REGION Network 9: Make Up Spin
   // Output if Throttle not disabled after a shift, flush not disabled, Drill Throttle Input Zero
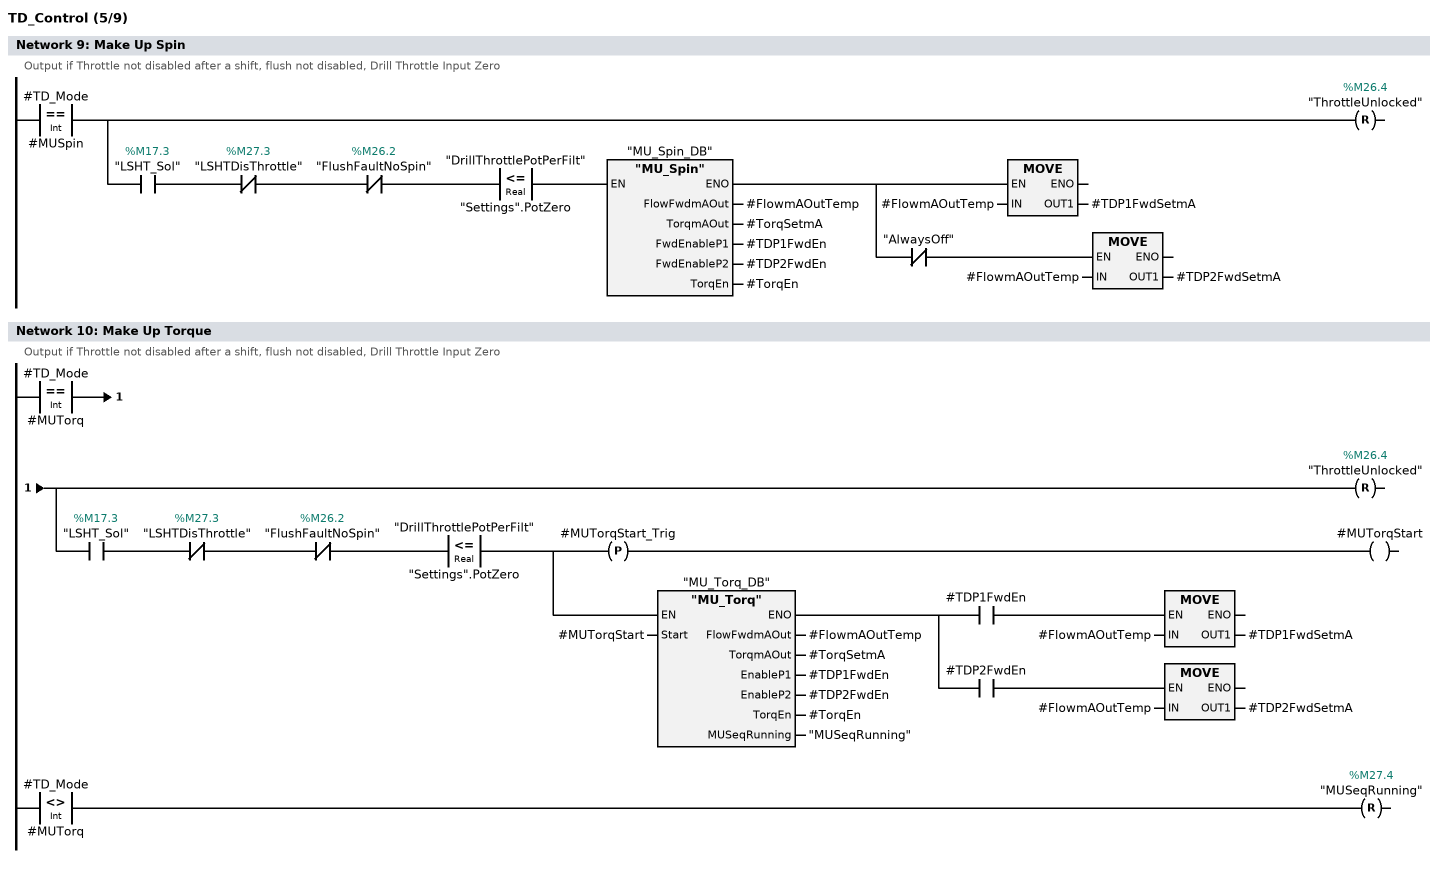
   RUNG wire#powerrail
      { S7_Templates := "SrcType := Int" } EQ_Contact(in1 := #TD_Mode, in2 := #MUSpin)
      wire#w1
      R_Coil( "ThrottleUnlocked" )
   END_RUNG
   RUNG wire#w1
      Contact( "LSHT_Sol" )
      I_Contact( "LSHTDisThrottle" )
      I_Contact( "FlushFaultNoSpin" )
      { S7_Templates := "SrcType := Real" } LE_Contact(in1 := "DrillThrottlePotPerFilt", in2 := "Settings".PotZero)
      "MU_Spin_DB"(FlowFwdmAOut => #FlowmAOutTemp, TorqmAOut => #TorqSetmA, FwdEnableP1 => #TDP1FwdEn, FwdEnableP2 => #TDP2FwdEn, TorqEn => #TorqEn)
      wire#w2
      Move(in := #FlowmAOutTemp, out1 => #TDP1FwdSetmA)
   END_RUNG
   RUNG wire#w2
      I_Contact( "AlwaysOff" )
      Move(in := #FlowmAOutTemp, out1 => #TDP2FwdSetmA)
   END_RUNG
   // the same network as SCL:
   #_w1 := #TD_Mode = #MUSpin;
   IF #_w1 THEN "ThrottleUnlocked" := FALSE; END_IF;
   "MU_Spin_DB"(EN := #_w1 AND "LSHT_Sol" AND NOT "LSHTDisThrottle" AND NOT "FlushFaultNoSpin" AND ("DrillThrottlePotPerFilt" <= "Settings".PotZero),   // "MU_Spin"
                FlowFwdmAOut => #FlowmAOutTemp,
                TorqmAOut => #TorqSetmA,
                FwdEnableP1 => #TDP1FwdEn,
                FwdEnableP2 => #TDP2FwdEn,
                TorqEn => #TorqEn,
                ENO => #_w2);
   IF #_w2 THEN #TDP1FwdSetmA := #FlowmAOutTemp; END_IF;
   IF #_w2 AND NOT "AlwaysOff" THEN #TDP2FwdSetmA := #FlowmAOutTemp; END_IF;
END_REGION

REGION Network 10: Make Up Torque
   // Output if Throttle not disabled after a shift, flush not disabled, Drill Throttle Input Zero
   RUNG wire#powerrail
      { S7_Templates := "SrcType := Int" } EQ_Contact(in1 := #TD_Mode, in2 := #MUTorq)
      wire#w1
      R_Coil( "ThrottleUnlocked" )
   END_RUNG
   RUNG wire#w1
      Contact( "LSHT_Sol" )
      I_Contact( "LSHTDisThrottle" )
      I_Contact( "FlushFaultNoSpin" )
      { S7_Templates := "SrcType := Real" } LE_Contact(in1 := "DrillThrottlePotPerFilt", in2 := "Settings".PotZero)
      wire#w2
      P_Trig( #MUTorqStart_Trig )
      Coil( #MUTorqStart )
   END_RUNG
   RUNG wire#w2
      "MU_Torq_DB"(Start := #MUTorqStart, FlowFwdmAOut => #FlowmAOutTemp, TorqmAOut => #TorqSetmA, EnableP1 => #TDP1FwdEn, EnableP2 => #TDP2FwdEn, TorqEn => #TorqEn, MUSeqRunning => "MUSeqRunning")
      wire#w3
      Contact( #TDP1FwdEn )
      Move(in := #FlowmAOutTemp, out1 => #TDP1FwdSetmA)
   END_RUNG
   RUNG wire#w3
      Contact( #TDP2FwdEn )
      Move(in := #FlowmAOutTemp, out1 => #TDP2FwdSetmA)
   END_RUNG
   RUNG wire#powerrail
      { S7_Templates := "SrcType := Int" } NE_Contact(in1 := #TD_Mode, in2 := #MUTorq)
      R_Coil( "MUSeqRunning" )
   END_RUNG
   // the same network as SCL:
   #_w1 := #TD_Mode = #MUTorq;
   IF #_w1 THEN "ThrottleUnlocked" := FALSE; END_IF;
   #_w2 := #_w1 AND "LSHT_Sol" AND NOT "LSHTDisThrottle" AND NOT "FlushFaultNoSpin" AND ("DrillThrottlePotPerFilt" <= "Settings".PotZero);
   #_w3 := #_w2 AND NOT #MUTorqStart_Trig;   // rising edge
   #MUTorqStart_Trig := #_w2;
   #MUTorqStart := #_w3;
   "MU_Torq_DB"(EN := #_w2,   // "MU_Torq"
                Start := #MUTorqStart,
                FlowFwdmAOut => #FlowmAOutTemp,
                TorqmAOut => #TorqSetmA,
                EnableP1 => #TDP1FwdEn,
                EnableP2 => #TDP2FwdEn,
                TorqEn => #TorqEn,
                MUSeqRunning => "MUSeqRunning",
                ENO => #_w4);
   IF #_w4 AND #TDP1FwdEn THEN #TDP1FwdSetmA := #FlowmAOutTemp; END_IF;
   IF #_w4 AND #TDP2FwdEn THEN #TDP2FwdSetmA := #FlowmAOutTemp; END_IF;
   IF #TD_Mode <> #MUTorq THEN "MUSeqRunning" := FALSE; END_IF;
END_REGION

REGION Network 11: Break Out
   // Output if Throttle not disabled after a shift, flush not disabled, Drill Throttle Input Zero.
   // No torq control in reverse. Set at relief
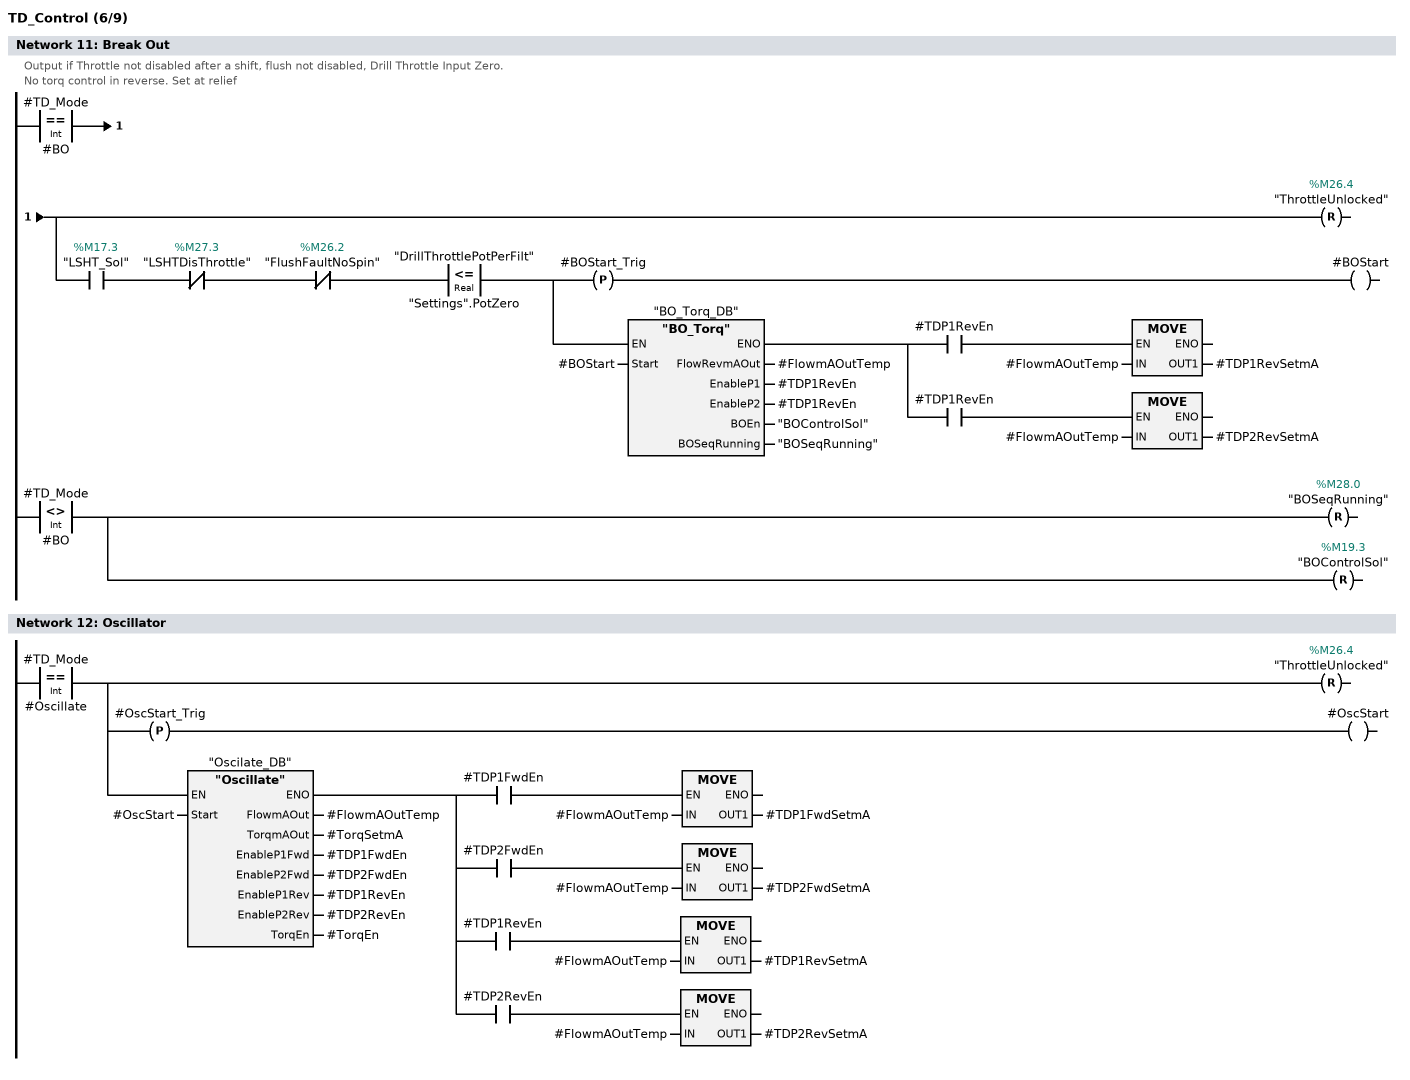
   RUNG wire#powerrail
      { S7_Templates := "SrcType := Int" } EQ_Contact(in1 := #TD_Mode, in2 := #BO)
      wire#w1
      R_Coil( "ThrottleUnlocked" )
   END_RUNG
   RUNG wire#w1
      Contact( "LSHT_Sol" )
      I_Contact( "LSHTDisThrottle" )
      I_Contact( "FlushFaultNoSpin" )
      { S7_Templates := "SrcType := Real" } LE_Contact(in1 := "DrillThrottlePotPerFilt", in2 := "Settings".PotZero)
      wire#w2
      P_Trig( #BOStart_Trig )
      Coil( #BOStart )
   END_RUNG
   RUNG wire#w2
      "BO_Torq_DB"(Start := #BOStart, FlowRevmAOut => #FlowmAOutTemp, EnableP1 => #TDP1RevEn, EnableP2 => #TDP1RevEn, BOEn => "BOControlSol", BOSeqRunning => "BOSeqRunning")
      wire#w3
      Contact( #TDP1RevEn )
      Move(in := #FlowmAOutTemp, out1 => #TDP1RevSetmA)
   END_RUNG
   RUNG wire#w3
      Contact( #TDP1RevEn )
      Move(in := #FlowmAOutTemp, out1 => #TDP2RevSetmA)
   END_RUNG
   RUNG wire#powerrail
      { S7_Templates := "SrcType := Int" } NE_Contact(in1 := #TD_Mode, in2 := #BO)
      wire#w4
      R_Coil( "BOSeqRunning" )
   END_RUNG
   RUNG wire#w4
      R_Coil( "BOControlSol" )
   END_RUNG
   // the same network as SCL:
   #_w1 := #TD_Mode = #BO;
   IF #_w1 THEN "ThrottleUnlocked" := FALSE; END_IF;
   #_w2 := #_w1 AND "LSHT_Sol" AND NOT "LSHTDisThrottle" AND NOT "FlushFaultNoSpin" AND ("DrillThrottlePotPerFilt" <= "Settings".PotZero);
   #_w3 := #_w2 AND NOT #BOStart_Trig;   // rising edge
   #BOStart_Trig := #_w2;
   #BOStart := #_w3;
   "BO_Torq_DB"(EN := #_w2,   // "BO_Torq"
                Start := #BOStart,
                FlowRevmAOut => #FlowmAOutTemp,
                EnableP1 => #TDP1RevEn,
                EnableP2 => #TDP1RevEn,
                BOEn => "BOControlSol",
                BOSeqRunning => "BOSeqRunning",
                ENO => #_w4);
   IF #_w4 AND #TDP1RevEn THEN
       #TDP1RevSetmA := #FlowmAOutTemp;
       #TDP2RevSetmA := #FlowmAOutTemp;
   END_IF;
   IF #TD_Mode <> #BO THEN
       "BOSeqRunning" := FALSE;
       "BOControlSol" := FALSE;
   END_IF;
END_REGION

REGION Network 12: Oscillator
   RUNG wire#powerrail
      { S7_Templates := "SrcType := Int" } EQ_Contact(in1 := #TD_Mode, in2 := #Oscillate)
      wire#w1
      R_Coil( "ThrottleUnlocked" )
   END_RUNG
   RUNG wire#w1
      P_Trig( #OscStart_Trig )
      Coil( #OscStart )
   END_RUNG
   RUNG wire#w1
      "Oscilate_DB"(Start := #OscStart, FlowmAOut => #FlowmAOutTemp, TorqmAOut => #TorqSetmA, EnableP1Fwd => #TDP1FwdEn, EnableP2Fwd => #TDP2FwdEn, EnableP1Rev => #TDP1RevEn, EnableP2Rev => #TDP2RevEn, TorqEn => #TorqEn)
      wire#w2
      Contact( #TDP1FwdEn )
      Move(in := #FlowmAOutTemp, out1 => #TDP1FwdSetmA)
   END_RUNG
   RUNG wire#w2
      Contact( #TDP2FwdEn )
      Move(in := #FlowmAOutTemp, out1 => #TDP2FwdSetmA)
   END_RUNG
   RUNG wire#w2
      Contact( #TDP1RevEn )
      Move(in := #FlowmAOutTemp, out1 => #TDP1RevSetmA)
   END_RUNG
   RUNG wire#w2
      Contact( #TDP2RevEn )
      Move(in := #FlowmAOutTemp, out1 => #TDP2RevSetmA)
   END_RUNG
   // the same network as SCL:
   #_w1 := #TD_Mode = #Oscillate;
   IF #_w1 THEN "ThrottleUnlocked" := FALSE; END_IF;
   #_w2 := #_w1 AND NOT #OscStart_Trig;   // rising edge
   #OscStart_Trig := #_w1;
   #OscStart := #_w2;
   "Oscilate_DB"(EN := #_w1,   // "Oscillate"
                 Start := #OscStart,
                 FlowmAOut => #FlowmAOutTemp,
                 TorqmAOut => #TorqSetmA,
                 EnableP1Fwd => #TDP1FwdEn,
                 EnableP2Fwd => #TDP2FwdEn,
                 EnableP1Rev => #TDP1RevEn,
                 EnableP2Rev => #TDP2RevEn,
                 TorqEn => #TorqEn,
                 ENO => #_w3);
   IF #_w3 AND #TDP1FwdEn THEN #TDP1FwdSetmA := #FlowmAOutTemp; END_IF;
   IF #_w3 AND #TDP2FwdEn THEN #TDP2FwdSetmA := #FlowmAOutTemp; END_IF;
   IF #_w3 AND #TDP1RevEn THEN #TDP1RevSetmA := #FlowmAOutTemp; END_IF;
   IF #_w3 AND #TDP2RevEn THEN #TDP2RevSetmA := #FlowmAOutTemp; END_IF;
END_REGION

REGION Network 13: Bypass Mode
   // In Bypass Mode
   // If gripper closed turn on Bypass valve(Quill is Locked after PTO funtioned)
   // After PTO wait 8 seconds for system to enage before enabling bypass control outputs
   // Note TD in HSLT in Bypass mode
   // Bypass Running flag will stay on for Set time after Bypass mode finished
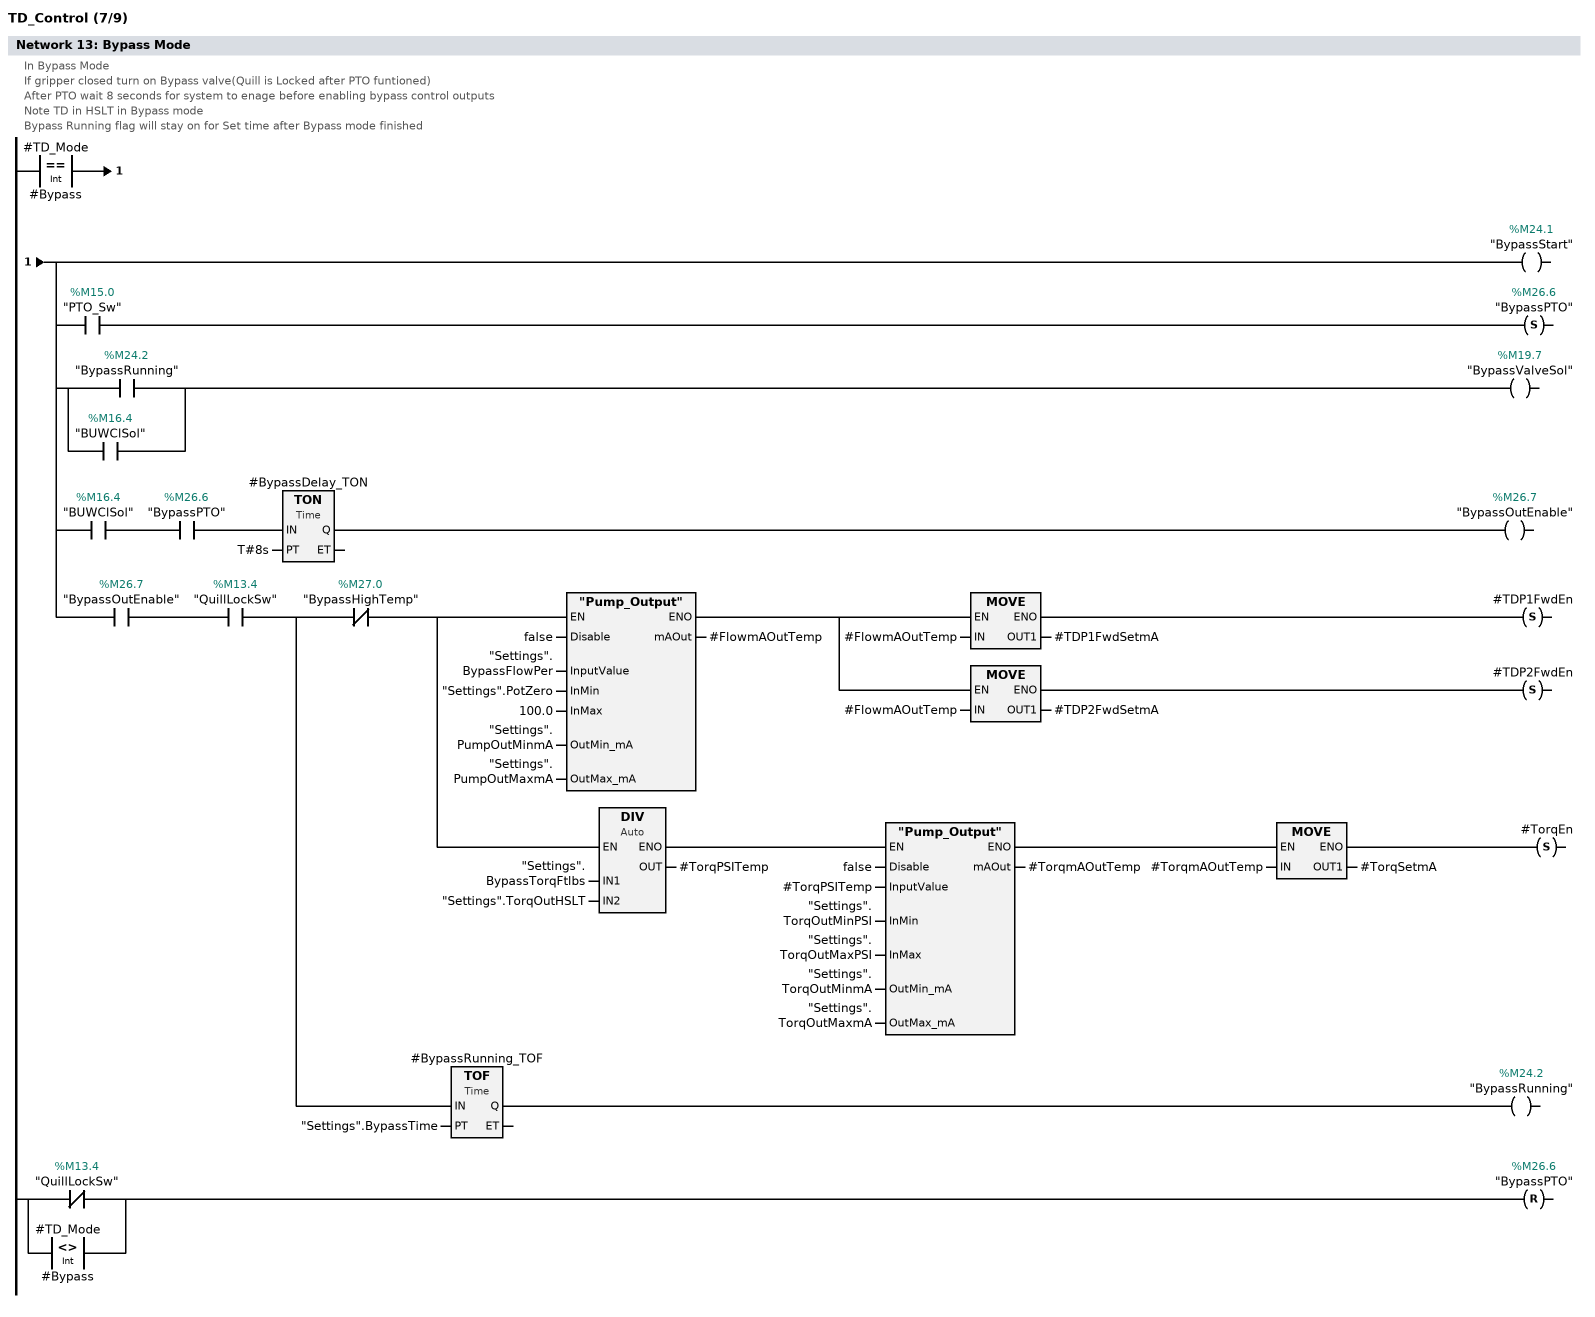
   RUNG wire#powerrail
      { S7_Templates := "SrcType := Int" } EQ_Contact(in1 := #TD_Mode, in2 := #Bypass)
      wire#w1
      Coil( "BypassStart" )
   END_RUNG
   RUNG wire#w1
      Contact( "PTO_Sw" )
      S_Coil( "BypassPTO" )
   END_RUNG
   RUNG wire#w1
      Contact( "BypassRunning" )
      wire#w2
      Coil( "BypassValveSol" )
   END_RUNG
   RUNG wire#w1
      Contact( "BUWClSol" )
   END_RUNG wire#w2
   RUNG wire#w1
      Contact( "BUWClSol" )
      Contact( "BypassPTO" )
      { S7_Templates := "time_type := Time" } #BypassDelay_TON.TON(pt := T#8s, et =>)
      Coil( "BypassOutEnable" )
   END_RUNG
   RUNG wire#w1
      Contact( "BypassOutEnable" )
      Contact( "QuillLockSw" )
      wire#w3
      I_Contact( "BypassHighTemp" )
      wire#w4
      "Pump_Output"(Disable := false, InputValue := "Settings".BypassFlowPer, InMin := "Settings".PotZero, InMax := 100.0, OutMin_mA := "Settings".PumpOutMinmA, OutMax_mA := "Settings".PumpOutMaxmA, mAOut => #FlowmAOutTemp)
      wire#w5
      Move(in := #FlowmAOutTemp, out1 => #TDP1FwdSetmA)
      S_Coil( #TDP1FwdEn )
   END_RUNG
   RUNG wire#w5
      Move(in := #FlowmAOutTemp, out1 => #TDP2FwdSetmA)
      S_Coil( #TDP2FwdEn )
   END_RUNG
   RUNG wire#w4
      Div(in1 := "Settings".BypassTorqFtlbs, in2 := "Settings".TorqOutHSLT, out => #TorqPSITemp)
      "Pump_Output"(Disable := false, InputValue := #TorqPSITemp, InMin := "Settings".TorqOutMinPSI, InMax := "Settings".TorqOutMaxPSI, OutMin_mA := "Settings".TorqOutMinmA, OutMax_mA := "Settings".TorqOutMaxmA, mAOut => #TorqmAOutTemp)
      Move(in := #TorqmAOutTemp, out1 => #TorqSetmA)
      S_Coil( #TorqEn )
   END_RUNG
   RUNG wire#w3
      { S7_Templates := "time_type := Time" } #BypassRunning_TOF.TOF(pt := "Settings".BypassTime, et =>)
      Coil( "BypassRunning" )
   END_RUNG
   RUNG wire#powerrail
      I_Contact( "QuillLockSw" )
      wire#w6
      R_Coil( "BypassPTO" )
   END_RUNG
   RUNG wire#powerrail
      { S7_Templates := "SrcType := Int" } NE_Contact(in1 := #TD_Mode, in2 := #Bypass)
   END_RUNG wire#w6
   // the same network as SCL:
   "BypassStart" := #TD_Mode = #Bypass;
   IF "BypassStart" AND "PTO_Sw" THEN "BypassPTO" := TRUE; END_IF;
   "BypassValveSol" := "BypassStart" AND ("BypassRunning" OR "BUWClSol");
   #BypassDelay_TON(IN := "BypassStart" AND "BUWClSol" AND "BypassPTO", PT := T#8s);   // TON
   "BypassOutEnable" := #BypassDelay_TON.Q;
   #_w1 := "BypassStart" AND "BypassOutEnable" AND "QuillLockSw";
   #_w3 := #_w1 AND NOT "BypassHighTemp";
   "Pump_Output"(EN := #_w1 AND NOT "BypassHighTemp",
                 Disable := false,
                 InputValue := "Settings".BypassFlowPer,
                 InMin := "Settings".PotZero,
                 InMax := 100.0,
                 OutMin_mA := "Settings".PumpOutMinmA,
                 OutMax_mA := "Settings".PumpOutMaxmA,
                 mAOut => #FlowmAOutTemp,
                 ENO => #_w2);
   IF #_w2 THEN
       #TDP1FwdSetmA := #FlowmAOutTemp;
       #TDP1FwdEn := TRUE;
       #TDP2FwdSetmA := #FlowmAOutTemp;
       #TDP2FwdEn := TRUE;
   END_IF;
   IF #_w3 THEN #TorqPSITemp := "Settings".BypassTorqFtlbs / "Settings".TorqOutHSLT; END_IF;
   "Pump_Output"(EN := #_w3,
                 Disable := false,
                 InputValue := #TorqPSITemp,
                 InMin := "Settings".TorqOutMinPSI,
                 InMax := "Settings".TorqOutMaxPSI,
                 OutMin_mA := "Settings".TorqOutMinmA,
                 OutMax_mA := "Settings".TorqOutMaxmA,
                 mAOut => #TorqmAOutTemp,
                 ENO => #_w4);
   IF #_w4 THEN
       #TorqSetmA := #TorqmAOutTemp;
       #TorqEn := TRUE;
   END_IF;
   #BypassRunning_TOF(IN := #_w1, PT := "Settings".BypassTime);   // TOF
   "BypassRunning" := #BypassRunning_TOF.Q;
   IF NOT "QuillLockSw" OR (#TD_Mode <> #Bypass) THEN "BypassPTO" := FALSE; END_IF;
END_REGION

REGION Network 14: Max Speed Limiter
   // Limit Output to Pump if speed above Max Speed Low Setpoint
   // While Limiting, Destroke Output to pump if above Max Speed High Setpoint and increase if below
   // Note In HSLT, drill mode active and both pumps used
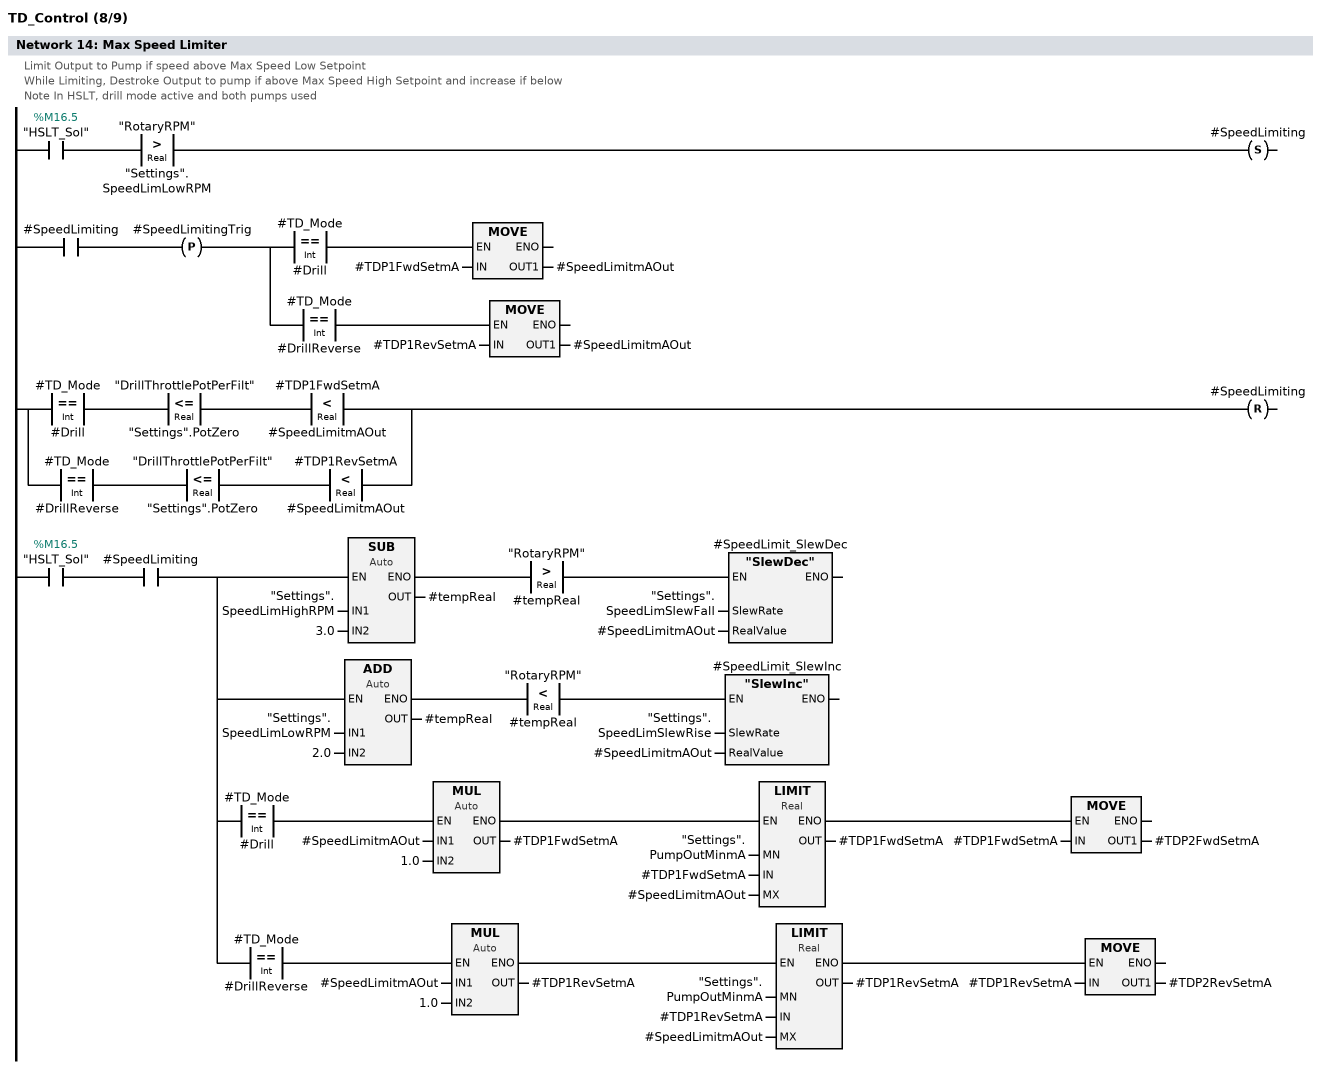
   RUNG wire#powerrail
      Contact( "HSLT_Sol" )
      { S7_Templates := "SrcType := Real" } GT_Contact(in1 := "RotaryRPM", in2 := "Settings".SpeedLimLowRPM)
      S_Coil( #SpeedLimiting )
   END_RUNG
   RUNG wire#powerrail
      Contact( #SpeedLimiting )
      P_Trig( #SpeedLimitingTrig )
      wire#w1
      { S7_Templates := "SrcType := Int" } EQ_Contact(in1 := #TD_Mode, in2 := #Drill)
      Move(in := #TDP1FwdSetmA, out1 => #SpeedLimitmAOut)
   END_RUNG
   RUNG wire#w1
      { S7_Templates := "SrcType := Int" } EQ_Contact(in1 := #TD_Mode, in2 := #DrillReverse)
      Move(in := #TDP1RevSetmA, out1 => #SpeedLimitmAOut)
   END_RUNG
   RUNG wire#powerrail
      { S7_Templates := "SrcType := Int" } EQ_Contact(in1 := #TD_Mode, in2 := #Drill)
      { S7_Templates := "SrcType := Real" } LE_Contact(in1 := "DrillThrottlePotPerFilt", in2 := "Settings".PotZero)
      { S7_Templates := "SrcType := Real" } LT_Contact(in1 := #TDP1FwdSetmA, in2 := #SpeedLimitmAOut)
      wire#w2
      R_Coil( #SpeedLimiting )
   END_RUNG
   RUNG wire#powerrail
      { S7_Templates := "SrcType := Int" } EQ_Contact(in1 := #TD_Mode, in2 := #DrillReverse)
      { S7_Templates := "SrcType := Real" } LE_Contact(in1 := "DrillThrottlePotPerFilt", in2 := "Settings".PotZero)
      { S7_Templates := "SrcType := Real" } LT_Contact(in1 := #TDP1RevSetmA, in2 := #SpeedLimitmAOut)
   END_RUNG wire#w2
   RUNG wire#powerrail
      Contact( "HSLT_Sol" )
      Contact( #SpeedLimiting )
      wire#w3
      Sub(in1 := "Settings".SpeedLimHighRPM, in2 := 3.0, out => #tempReal)
      { S7_Templates := "SrcType := Real" } GT_Contact(in1 := "RotaryRPM", in2 := #tempReal)
      #SpeedLimit_SlewDec(SlewRate := "Settings".SpeedLimSlewFall, RealValue := #SpeedLimitmAOut)
   END_RUNG
   RUNG wire#w3
      Add(in1 := "Settings".SpeedLimLowRPM, in2 := 2.0, out => #tempReal)
      { S7_Templates := "SrcType := Real" } LT_Contact(in1 := "RotaryRPM", in2 := #tempReal)
      #SpeedLimit_SlewInc(SlewRate := "Settings".SpeedLimSlewRise, RealValue := #SpeedLimitmAOut)
   END_RUNG
   RUNG wire#w3
      { S7_Templates := "SrcType := Int" } EQ_Contact(in1 := #TD_Mode, in2 := #Drill)
      Mul(in1 := #SpeedLimitmAOut, in2 := 1.0, out => #TDP1FwdSetmA)
      { S7_Templates := "value_type := Real" } Limit(mn := "Settings".PumpOutMinmA, in := #TDP1FwdSetmA, mx := #SpeedLimitmAOut, out => #TDP1FwdSetmA)
      Move(in := #TDP1FwdSetmA, out1 => #TDP2FwdSetmA)
   END_RUNG
   RUNG wire#w3
      { S7_Templates := "SrcType := Int" } EQ_Contact(in1 := #TD_Mode, in2 := #DrillReverse)
      Mul(in1 := #SpeedLimitmAOut, in2 := 1.0, out => #TDP1RevSetmA)
      { S7_Templates := "value_type := Real" } Limit(mn := "Settings".PumpOutMinmA, in := #TDP1RevSetmA, mx := #SpeedLimitmAOut, out => #TDP1RevSetmA)
      Move(in := #TDP1RevSetmA, out1 => #TDP2RevSetmA)
   END_RUNG
   // the same network as SCL:
   IF "HSLT_Sol" AND ("RotaryRPM" > "Settings".SpeedLimLowRPM) THEN #SpeedLimiting := TRUE; END_IF;
   #_w1 := #SpeedLimiting AND NOT #SpeedLimitingTrig;   // rising edge
   #SpeedLimitingTrig := #SpeedLimiting;
   IF #_w1 AND (#TD_Mode = #Drill) THEN #SpeedLimitmAOut := #TDP1FwdSetmA; END_IF;
   IF #_w1 AND (#TD_Mode = #DrillReverse) THEN #SpeedLimitmAOut := #TDP1RevSetmA; END_IF;
   IF ((#TD_Mode = #Drill) AND ("DrillThrottlePotPerFilt" <= "Settings".PotZero) AND (#TDP1FwdSetmA < #SpeedLimitmAOut)) OR ((#TD_Mode = #DrillReverse) AND ("DrillThrottlePotPerFilt" <= "Settings".PotZero) AND (#TDP1RevSetmA < #SpeedLimitmAOut)) THEN
       #SpeedLimiting := FALSE;
   END_IF;
   #_w2 := "HSLT_Sol" AND #SpeedLimiting;
   IF #_w2 THEN #tempReal := "Settings".SpeedLimHighRPM - 3.0; END_IF;
   IF #_w2 AND ("RotaryRPM" > #tempReal) THEN
       #SpeedLimit_SlewDec(SlewRate := "Settings".SpeedLimSlewFall, RealValue := #SpeedLimitmAOut);   // "SlewDec"
   END_IF;
   IF #_w2 THEN #tempReal := "Settings".SpeedLimLowRPM + 2.0; END_IF;
   IF #_w2 AND ("RotaryRPM" < #tempReal) THEN
       #SpeedLimit_SlewInc(SlewRate := "Settings".SpeedLimSlewRise, RealValue := #SpeedLimitmAOut);   // "SlewInc"
   END_IF;
   IF #_w2 AND (#TD_Mode = #Drill) THEN
       #TDP1FwdSetmA := #SpeedLimitmAOut * 1.0;
       #TDP1FwdSetmA := LIMIT(MN := "Settings".PumpOutMinmA, IN := #TDP1FwdSetmA, MX := #SpeedLimitmAOut);
       #TDP2FwdSetmA := #TDP1FwdSetmA;
   END_IF;
   IF #_w2 AND (#TD_Mode = #DrillReverse) THEN
       #TDP1RevSetmA := #SpeedLimitmAOut * 1.0;
       #TDP1RevSetmA := LIMIT(MN := "Settings".PumpOutMinmA, IN := #TDP1RevSetmA, MX := #SpeedLimitmAOut);
       #TDP2RevSetmA := #TDP1RevSetmA;
   END_IF;
END_REGION

REGION Network 15: High Temp Speed Limiter
   // Limit Flow mA Output if High Temp reduced RPM.
   // 
   // Disable outputs 10 seconds after a shutdown and disable Throttle
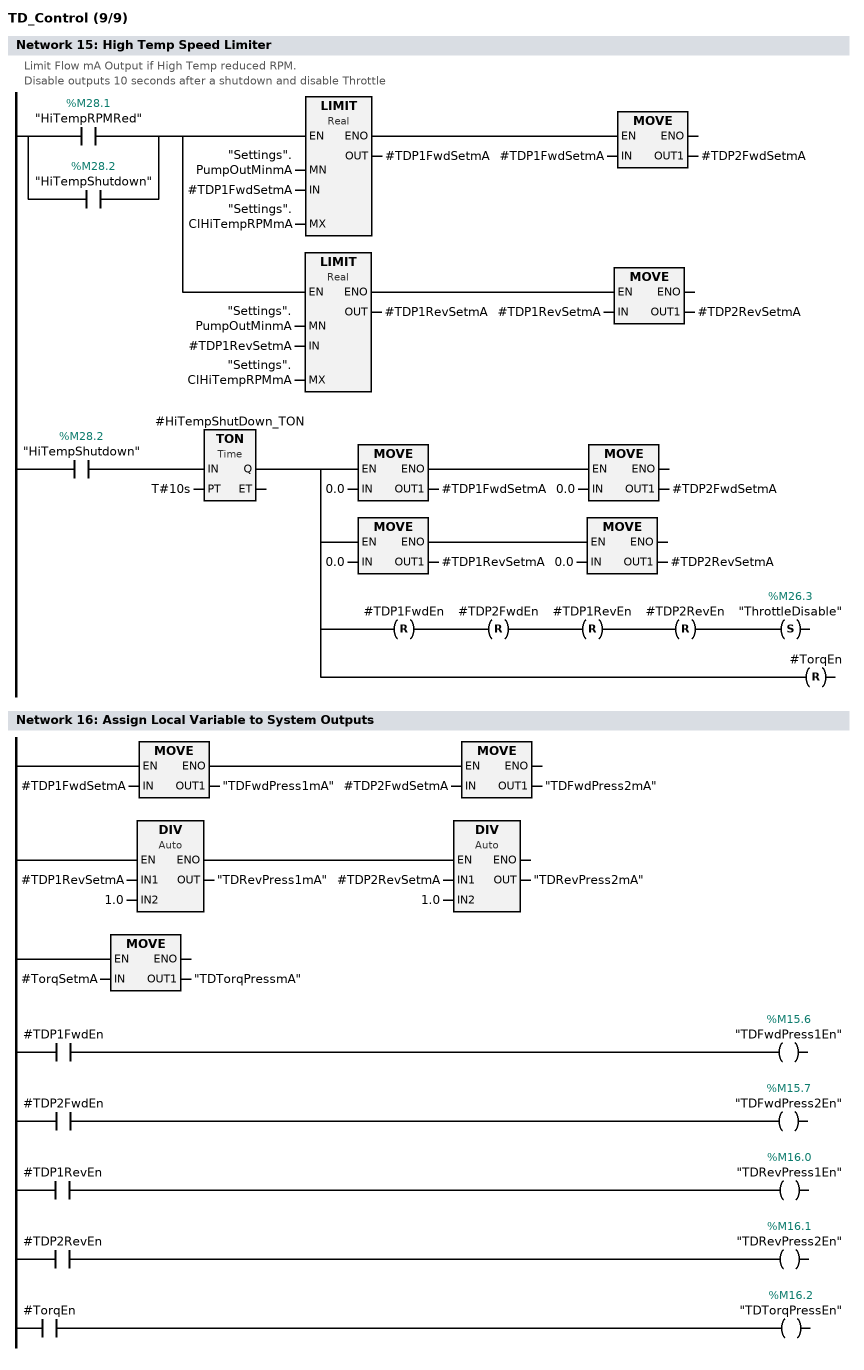
   RUNG wire#powerrail
      Contact( "HiTempRPMRed" )
      wire#w1
      { S7_Templates := "value_type := Real" } Limit(mn := "Settings".PumpOutMinmA, in := #TDP1FwdSetmA, mx := "Settings".ClHiTempRPMmA, out => #TDP1FwdSetmA)
      Move(in := #TDP1FwdSetmA, out1 => #TDP2FwdSetmA)
   END_RUNG
   RUNG wire#powerrail
      Contact( "HiTempShutdown" )
   END_RUNG wire#w1
   RUNG wire#w1
      { S7_Templates := "value_type := Real" } Limit(mn := "Settings".PumpOutMinmA, in := #TDP1RevSetmA, mx := "Settings".ClHiTempRPMmA, out => #TDP1RevSetmA)
      Move(in := #TDP1RevSetmA, out1 => #TDP2RevSetmA)
   END_RUNG
   RUNG wire#powerrail
      Contact( "HiTempShutdown" )
      { S7_Templates := "time_type := Time" } #HiTempShutDown_TON.TON(pt := T#10s, et =>)
      wire#w2
      Move(in := 0.0, out1 => #TDP1FwdSetmA)
      Move(in := 0.0, out1 => #TDP2FwdSetmA)
   END_RUNG
   RUNG wire#w2
      Move(in := 0.0, out1 => #TDP1RevSetmA)
      Move(in := 0.0, out1 => #TDP2RevSetmA)
   END_RUNG
   RUNG wire#w2
      R_Coil( #TDP1FwdEn )
      R_Coil( #TDP2FwdEn )
      R_Coil( #TDP1RevEn )
      R_Coil( #TDP2RevEn )
      S_Coil( "ThrottleDisable" )
   END_RUNG
   RUNG wire#w2
      R_Coil( #TorqEn )
   END_RUNG
   // the same network as SCL:
   IF "HiTempRPMRed" OR "HiTempShutdown" THEN
       #TDP1FwdSetmA := LIMIT(MN := "Settings".PumpOutMinmA, IN := #TDP1FwdSetmA, MX := "Settings".ClHiTempRPMmA);
       #TDP2FwdSetmA := #TDP1FwdSetmA;
       #TDP1RevSetmA := LIMIT(MN := "Settings".PumpOutMinmA, IN := #TDP1RevSetmA, MX := "Settings".ClHiTempRPMmA);
       #TDP2RevSetmA := #TDP1RevSetmA;
   END_IF;
   #HiTempShutDown_TON(IN := "HiTempShutdown", PT := T#10s);   // TON
   IF #HiTempShutDown_TON.Q THEN
       #TDP1FwdSetmA := 0.0;
       #TDP2FwdSetmA := 0.0;
       #TDP1RevSetmA := 0.0;
       #TDP2RevSetmA := 0.0;
       #TDP1FwdEn := FALSE;
       #TDP2FwdEn := FALSE;
       #TDP1RevEn := FALSE;
       #TDP2RevEn := FALSE;
       "ThrottleDisable" := TRUE;
       #TorqEn := FALSE;
   END_IF;
END_REGION

REGION Network 16: Assign Local Variable to System Outputs
   RUNG wire#powerrail
      Move(in := #TDP1FwdSetmA, out1 => "TDFwdPress1mA")
      Move(in := #TDP2FwdSetmA, out1 => "TDFwdPress2mA")
   END_RUNG
   RUNG wire#powerrail
      Div(in1 := #TDP1RevSetmA, in2 := 1.0, out => "TDRevPress1mA")
      Div(in1 := #TDP2RevSetmA, in2 := 1.0, out => "TDRevPress2mA")
   END_RUNG
   RUNG wire#powerrail
      Move(in := #TorqSetmA, out1 => "TDTorqPressmA")
   END_RUNG
   RUNG wire#powerrail
      Contact( #TDP1FwdEn )
      Coil( "TDFwdPress1En" )
   END_RUNG
   RUNG wire#powerrail
      Contact( #TDP2FwdEn )
      Coil( "TDFwdPress2En" )
   END_RUNG
   RUNG wire#powerrail
      Contact( #TDP1RevEn )
      Coil( "TDRevPress1En" )
   END_RUNG
   RUNG wire#powerrail
      Contact( #TDP2RevEn )
      Coil( "TDRevPress2En" )
   END_RUNG
   RUNG wire#powerrail
      Contact( #TorqEn )
      Coil( "TDTorqPressEn" )
   END_RUNG
   // the same network as SCL:
   "TDFwdPress1mA" := #TDP1FwdSetmA;
   "TDFwdPress2mA" := #TDP2FwdSetmA;
   "TDRevPress1mA" := #TDP1RevSetmA / 1.0;
   "TDRevPress2mA" := #TDP2RevSetmA / 1.0;
   "TDTorqPressmA" := #TorqSetmA;
   "TDFwdPress1En" := #TDP1FwdEn;
   "TDFwdPress2En" := #TDP2FwdEn;
   "TDRevPress1En" := #TDP1RevEn;
   "TDRevPress2En" := #TDP2RevEn;
   "TDTorqPressEn" := #TorqEn;
END_REGION
END_FUNCTION_BLOCK

FUNCTION_BLOCK "Drill"   // FB30, LAD
TITLE = Drill
{ S7_Optimized_Access := 'TRUE' }
// Written BY Kristopher Gimenez Feb 3,2023
// This block is used to control the TD Drill mode
// stored: AutoNumber false, MemoryReserve 100, SetENOAutomatically false
   VAR_INPUT
      DrillPSISet : Real;
      DisableThrottle : Bool;
   END_VAR
   VAR_OUTPUT
      FlowFwdmAOut : Real;
      FwdEnableP1 : Bool;
      TorquePSIOut : Real;
      FwdEnableP2 : Bool;
   END_VAR
   VAR
      PSinitialize : Bool := False;
      TorqLowLimitFtLbs { ExternalAccessible := 'False'; ExternalVisible := 'False'; ExternalWritable := 'False'} : Real;   // Above this value flow will be detroked
      TorqHighLimitFtLbs : Real;
      TorqLimiting : Bool;   // Bit to indicate torq limiting
      TorqLimitTrig : Bool;   // Bit used for positive trigger transition on Torq Limiting
      LimitFlowmAOut : Real;   // Calculated limited output value for flow
      TorqLimit_TON { S7_SetPoint := 'True'} : TON_TIME;
      TorqLimit_SlewDec { S7_SetPoint := 'True'} : "SlewDec";
      Torq_Limit_SlewInc { S7_SetPoint := 'True'} : "SlewInc";
   END_VAR
   VAR_TEMP
      PSIsetHIgh : Real;
      PSIsetLow : Real;
      PSIcheck : Real;
      PSiRange : Real;
      PSIadjustRange : Real;
      PSIadjustval : Real;
      PsiPos : Bool;
      PSIinitial : Bool;
      PSIAdjust : Bool;
      FlowmAOutTemp : Real;
      TempPSI : Real;
      tempReal : Real;
   END_VAR
   VAR_TEMP   // added for the SCL form of the ladder/FBD networks
      _w1 : Bool;
      _w2 : Bool;
      _w3 : Bool;
   END_VAR
BEGIN

REGION Network 1: Speed Setpoint
   // If throttle not disable get speed setpoint
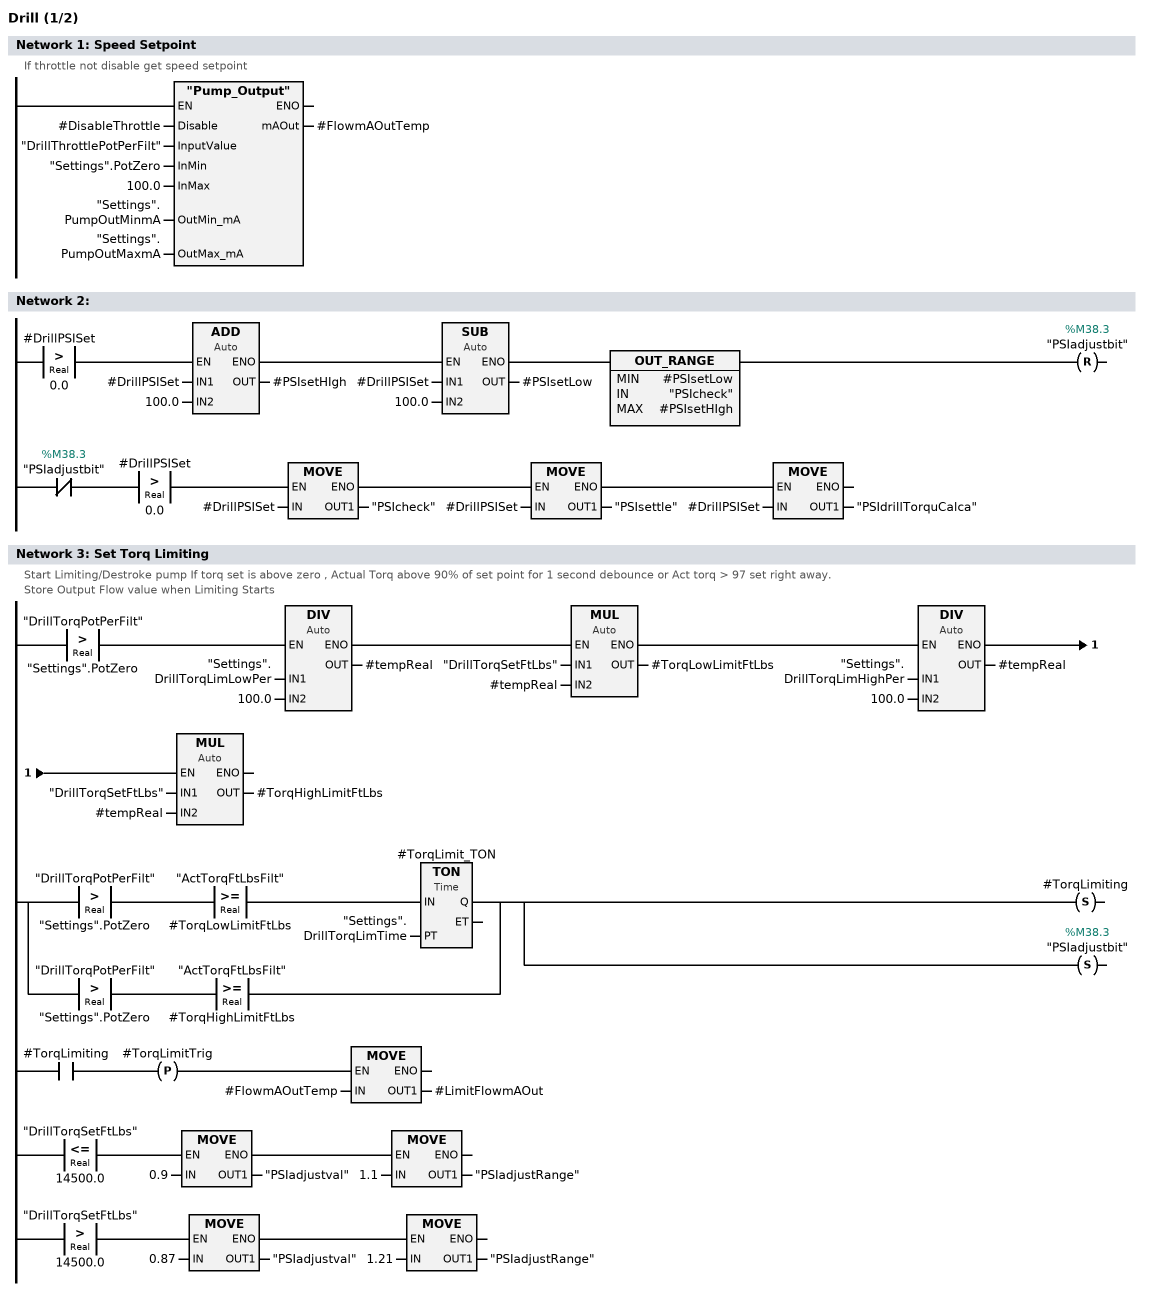
   RUNG wire#powerrail
      "Pump_Output"(Disable := #DisableThrottle, InputValue := "DrillThrottlePotPerFilt", InMin := "Settings".PotZero, InMax := 100.0, OutMin_mA := "Settings".PumpOutMinmA, OutMax_mA := "Settings".PumpOutMaxmA, mAOut => #FlowmAOutTemp)
   END_RUNG
   // the same network as SCL:
   "Pump_Output"(Disable := #DisableThrottle,
                 InputValue := "DrillThrottlePotPerFilt",
                 InMin := "Settings".PotZero,
                 InMax := 100.0,
                 OutMin_mA := "Settings".PumpOutMinmA,
                 OutMax_mA := "Settings".PumpOutMaxmA,
                 mAOut => #FlowmAOutTemp);
END_REGION

REGION Network 2
   #_w1 := #DrillPSISet > 0.0;
   IF #_w1 THEN
       #PSIsetHIgh := #DrillPSISet + 100.0;
       #PSIsetLow := #DrillPSISet - 100.0;
   END_IF;
   IF #_w1 AND (("PSIcheck" < #PSIsetLow) OR ("PSIcheck" > #PSIsetHIgh)) THEN
       "PSIadjustbit" := FALSE;
   END_IF;
   IF NOT "PSIadjustbit" AND (#DrillPSISet > 0.0) THEN
       "PSIcheck" := #DrillPSISet;
       "PSIsettle" := #DrillPSISet;
       "PSIdrillTorquCalca" := #DrillPSISet;
   END_IF;
END_REGION

REGION Network 3: Set Torq Limiting
   // Start Limiting/Destroke pump If torq set is above zero , Actual Torq above 90% of set point for 1 second debounce or Act torq > 97 set right away. 
   // Store Output Flow value when Limiting Starts
   RUNG wire#powerrail
      { S7_Templates := "SrcType := Real" } GT_Contact(in1 := "DrillTorqPotPerFilt", in2 := "Settings".PotZero)
      Div(in1 := "Settings".DrillTorqLimLowPer, in2 := 100.0, out => #tempReal)
      Mul(in1 := "DrillTorqSetFtLbs", in2 := #tempReal, out => #TorqLowLimitFtLbs)
      Div(in1 := "Settings".DrillTorqLimHighPer, in2 := 100.0, out => #tempReal)
      Mul(in1 := "DrillTorqSetFtLbs", in2 := #tempReal, out => #TorqHighLimitFtLbs)
   END_RUNG
   RUNG wire#powerrail
      { S7_Templates := "SrcType := Real" } GT_Contact(in1 := "DrillTorqPotPerFilt", in2 := "Settings".PotZero)
      { S7_Templates := "SrcType := Real" } GE_Contact(in1 := "ActTorqFtLbsFilt", in2 := #TorqLowLimitFtLbs)
      { S7_Templates := "time_type := Time" } #TorqLimit_TON.TON(pt := "Settings".DrillTorqLimTime, et =>)
      wire#w1
      S_Coil( #TorqLimiting )
   END_RUNG
   RUNG wire#powerrail
      { S7_Templates := "SrcType := Real" } GT_Contact(in1 := "DrillTorqPotPerFilt", in2 := "Settings".PotZero)
      { S7_Templates := "SrcType := Real" } GE_Contact(in1 := "ActTorqFtLbsFilt", in2 := #TorqHighLimitFtLbs)
   END_RUNG wire#w1
   RUNG wire#w1
      S_Coil( "PSIadjustbit" )
   END_RUNG
   RUNG wire#powerrail
      Contact( #TorqLimiting )
      P_Trig( #TorqLimitTrig )
      Move(in := #FlowmAOutTemp, out1 => #LimitFlowmAOut)
   END_RUNG
   RUNG wire#powerrail
      { S7_Templates := "SrcType := Real" } LE_Contact(in1 := "DrillTorqSetFtLbs", in2 := 14500.0)
      Move(in := 0.9, out1 => "PSIadjustval")
      Move(in := 1.1, out1 => "PSIadjustRange")
   END_RUNG
   RUNG wire#powerrail
      { S7_Templates := "SrcType := Real" } GT_Contact(in1 := "DrillTorqSetFtLbs", in2 := 14500.0)
      Move(in := 0.87, out1 => "PSIadjustval")
      Move(in := 1.21, out1 => "PSIadjustRange")
   END_RUNG
   // the same network as SCL:
   IF "DrillTorqPotPerFilt" > "Settings".PotZero THEN
       #tempReal := "Settings".DrillTorqLimLowPer / 100.0;
       #TorqLowLimitFtLbs := "DrillTorqSetFtLbs" * #tempReal;
       #tempReal := "Settings".DrillTorqLimHighPer / 100.0;
       #TorqHighLimitFtLbs := "DrillTorqSetFtLbs" * #tempReal;
   END_IF;
   #TorqLimit_TON(IN := ("DrillTorqPotPerFilt" > "Settings".PotZero) AND ("ActTorqFtLbsFilt" >= #TorqLowLimitFtLbs),   // TON
                  PT := "Settings".DrillTorqLimTime);
   IF #TorqLimit_TON.Q OR (("DrillTorqPotPerFilt" > "Settings".PotZero) AND ("ActTorqFtLbsFilt" >= #TorqHighLimitFtLbs)) THEN
       #TorqLimiting := TRUE;
       "PSIadjustbit" := TRUE;
   END_IF;
   #_w1 := #TorqLimiting AND NOT #TorqLimitTrig;   // rising edge
   #TorqLimitTrig := #TorqLimiting;
   IF #_w1 THEN #LimitFlowmAOut := #FlowmAOutTemp; END_IF;
   IF "DrillTorqSetFtLbs" <= 14500.0 THEN
       "PSIadjustval" := 0.9;
       "PSIadjustRange" := 1.1;
   END_IF;
   IF "DrillTorqSetFtLbs" > 14500.0 THEN
       "PSIadjustval" := 0.87;
       "PSIadjustRange" := 1.21;
   END_IF;
END_REGION

REGION Network 4: Flow Control in Torq Limit
   // If torq limiting-
   // in High torq  destroke the ouput. 
   // - if low torq increase stroke back to setpoint
   // -Otherwise hold.  
   // Slew rate are mA/sec. TON increment set to 10ms so unput Slew rate divided by 100
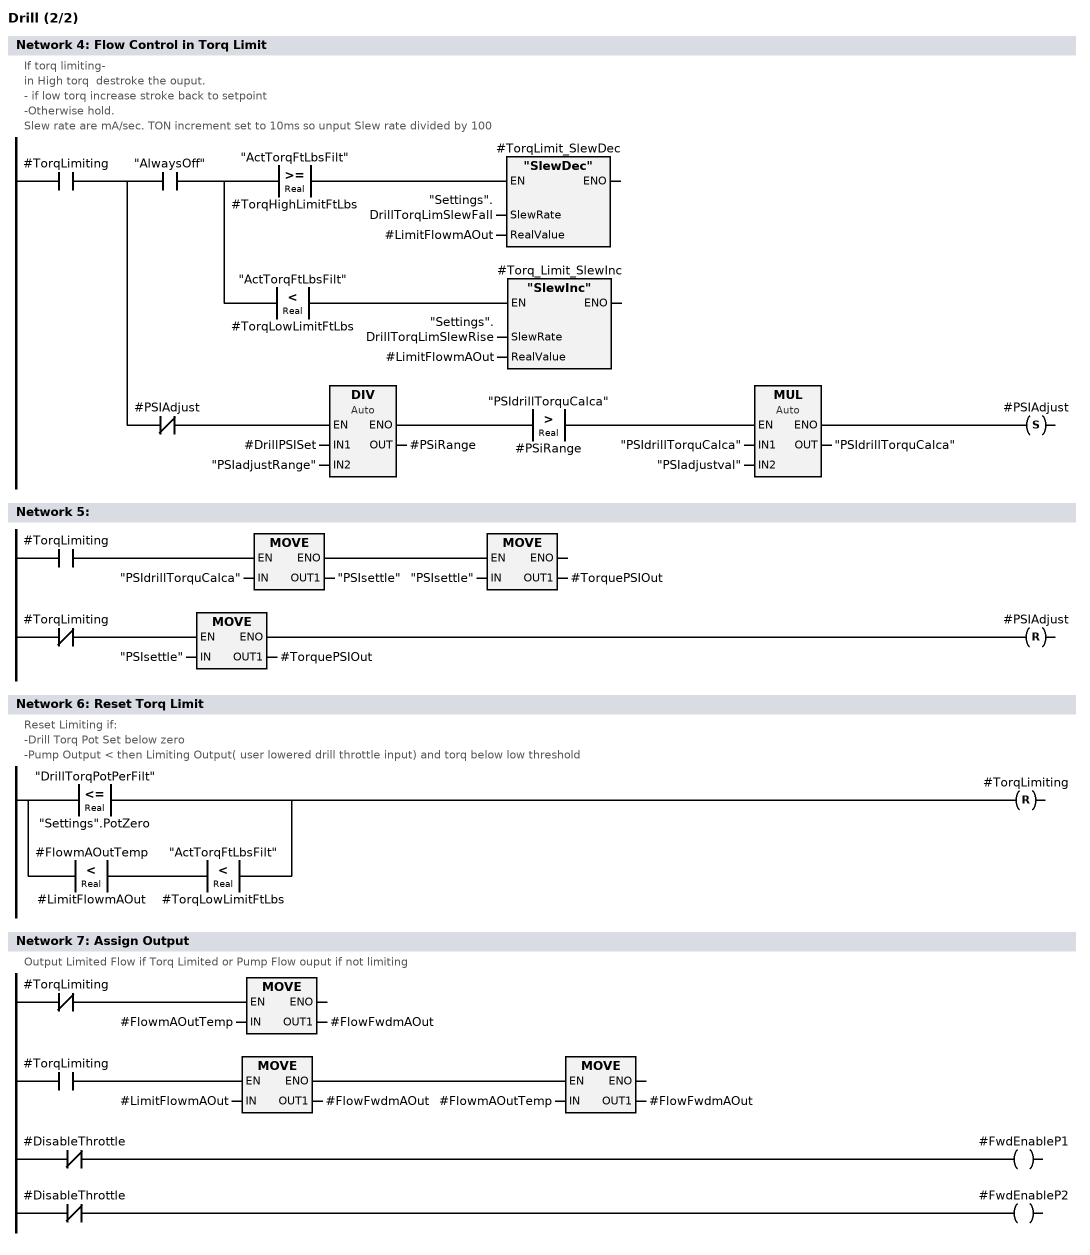
   RUNG wire#powerrail
      Contact( #TorqLimiting )
      wire#w1
      Contact( "AlwaysOff" )
      wire#w2
      { S7_Templates := "SrcType := Real" } GE_Contact(in1 := "ActTorqFtLbsFilt", in2 := #TorqHighLimitFtLbs)
      #TorqLimit_SlewDec(SlewRate := "Settings".DrillTorqLimSlewFall, RealValue := #LimitFlowmAOut)
   END_RUNG
   RUNG wire#w2
      { S7_Templates := "SrcType := Real" } LT_Contact(in1 := "ActTorqFtLbsFilt", in2 := #TorqLowLimitFtLbs)
      #Torq_Limit_SlewInc(SlewRate := "Settings".DrillTorqLimSlewRise, RealValue := #LimitFlowmAOut)
   END_RUNG
   RUNG wire#w1
      I_Contact( #PSIAdjust )
      Div(in1 := #DrillPSISet, in2 := "PSIadjustRange", out => #PSiRange)
      { S7_Templates := "SrcType := Real" } GT_Contact(in1 := "PSIdrillTorquCalca", in2 := #PSiRange)
      Mul(in1 := "PSIdrillTorquCalca", in2 := "PSIadjustval", out => "PSIdrillTorquCalca")
      S_Coil( #PSIAdjust )
   END_RUNG
   // the same network as SCL:
   #_w1 := #TorqLimiting AND "AlwaysOff";
   IF #_w1 AND ("ActTorqFtLbsFilt" >= #TorqHighLimitFtLbs) THEN
       #TorqLimit_SlewDec(SlewRate := "Settings".DrillTorqLimSlewFall, RealValue := #LimitFlowmAOut);   // "SlewDec"
   END_IF;
   IF #_w1 AND ("ActTorqFtLbsFilt" < #TorqLowLimitFtLbs) THEN
       #Torq_Limit_SlewInc(SlewRate := "Settings".DrillTorqLimSlewRise, RealValue := #LimitFlowmAOut);   // "SlewInc"
   END_IF;
   #_w2 := #TorqLimiting AND NOT #PSIAdjust;
   IF #_w2 THEN #PSiRange := #DrillPSISet / "PSIadjustRange"; END_IF;
   #_w3 := #_w2 AND ("PSIdrillTorquCalca" > #PSiRange);
   IF #_w3 THEN
       "PSIdrillTorquCalca" := "PSIdrillTorquCalca" * "PSIadjustval";
       #PSIAdjust := TRUE;
   END_IF;
END_REGION

REGION Network 5
   RUNG wire#powerrail
      Contact( #TorqLimiting )
      Move(in := "PSIdrillTorquCalca", out1 => "PSIsettle")
      Move(in := "PSIsettle", out1 => #TorquePSIOut)
   END_RUNG
   RUNG wire#powerrail
      I_Contact( #TorqLimiting )
      Move(in := "PSIsettle", out1 => #TorquePSIOut)
      R_Coil( #PSIAdjust )
   END_RUNG
   // the same network as SCL:
   IF #TorqLimiting THEN
       "PSIsettle" := "PSIdrillTorquCalca";
       #TorquePSIOut := "PSIsettle";
   END_IF;
   IF NOT #TorqLimiting THEN
       #TorquePSIOut := "PSIsettle";
       #PSIAdjust := FALSE;
   END_IF;
END_REGION

REGION Network 6: Reset Torq Limit
   // Reset Limiting if:
   // -Drill Torq Pot Set below zero
   //  -Pump Output < then Limiting Output( user lowered drill throttle input) and torq below low threshold
   RUNG wire#powerrail
      { S7_Templates := "SrcType := Real" } LE_Contact(in1 := "DrillTorqPotPerFilt", in2 := "Settings".PotZero)
      wire#w1
      R_Coil( #TorqLimiting )
   END_RUNG
   RUNG wire#powerrail
      { S7_Templates := "SrcType := Real" } LT_Contact(in1 := #FlowmAOutTemp, in2 := #LimitFlowmAOut)
      { S7_Templates := "SrcType := Real" } LT_Contact(in1 := "ActTorqFtLbsFilt", in2 := #TorqLowLimitFtLbs)
   END_RUNG wire#w1
   // the same network as SCL:
   IF ("DrillTorqPotPerFilt" <= "Settings".PotZero) OR ((#FlowmAOutTemp < #LimitFlowmAOut) AND ("ActTorqFtLbsFilt" < #TorqLowLimitFtLbs)) THEN
       #TorqLimiting := FALSE;
   END_IF;
END_REGION

REGION Network 7: Assign Output
   // Output Limited Flow if Torq Limited or Pump Flow ouput if not limiting
   RUNG wire#powerrail
      I_Contact( #TorqLimiting )
      Move(in := #FlowmAOutTemp, out1 => #FlowFwdmAOut)
   END_RUNG
   RUNG wire#powerrail
      Contact( #TorqLimiting )
      Move(in := #LimitFlowmAOut, out1 => #FlowFwdmAOut)
      Move(in := #FlowmAOutTemp, out1 => #FlowFwdmAOut)
   END_RUNG
   RUNG wire#powerrail
      I_Contact( #DisableThrottle )
      Coil( #FwdEnableP1 )
   END_RUNG
   RUNG wire#powerrail
      I_Contact( #DisableThrottle )
      Coil( #FwdEnableP2 )
   END_RUNG
   // the same network as SCL:
   IF NOT #TorqLimiting THEN #FlowFwdmAOut := #FlowmAOutTemp; END_IF;
   IF #TorqLimiting THEN
       #FlowFwdmAOut := #LimitFlowmAOut;
       #FlowFwdmAOut := #FlowmAOutTemp;
   END_IF;
   #FwdEnableP1 := NOT #DisableThrottle;
   #FwdEnableP2 := NOT #DisableThrottle;
END_REGION
END_FUNCTION_BLOCK

FUNCTION_BLOCK "SlewDec"   // FB123, LAD
TITLE = SlewInc
{ S7_Optimized_Access := 'TRUE' }
// Written BY Kristopher Gimenez Feb 17th ,2023
// This block will be used to slew the output but the at the set rate per second base on input slew rate
// stored: AutoNumber false, MemoryReserve 100, SetENOAutomatically false
   VAR_INPUT
      SlewRate : Real;   // Slew rate in mA/sec
   END_VAR
   VAR_IN_OUT
      RealValue : Real;
   END_VAR
   VAR
      Slew : Bool;
      Dec_TON : TON_TIME;
   END_VAR
   VAR_TEMP
      tempReal : Real;
   END_VAR
BEGIN

REGION Network 1: Slew rate in mA/sec
   // Decrease the input value by the slew rate
   // Decreasing every 10ms divide rate by 100
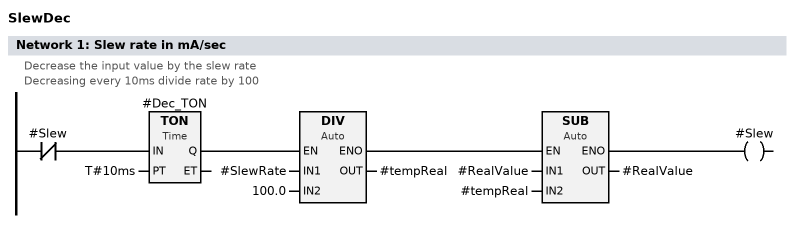
   RUNG wire#powerrail
      I_Contact( #Slew )
      { S7_Templates := "time_type := Time" } #Dec_TON.TON(pt := T#10ms, et =>)
      Div(in1 := #SlewRate, in2 := 100.0, out => #tempReal)
      Sub(in1 := #RealValue, in2 := #tempReal, out => #RealValue)
      Coil( #Slew )
   END_RUNG
   // the same network as SCL:
   #Dec_TON(IN := NOT #Slew, PT := T#10ms);   // TON
   IF #Dec_TON.Q THEN
       #tempReal := #SlewRate / 100.0;
       #RealValue := #RealValue - #tempReal;
   END_IF;
   #Slew := #Dec_TON.Q;
END_REGION
END_FUNCTION_BLOCK

FUNCTION_BLOCK "SlewInc"   // FB122, LAD
TITLE = SlewInc
{ S7_Optimized_Access := 'TRUE' }
// Written BY Kristopher Gimenez Feb 17,2023
// This block will be used to slew the output but the at the set rate per second base on input slew rate
// stored: AutoNumber false, MemoryReserve 100, SetENOAutomatically false
   VAR_INPUT
      SlewRate : Real;   // Slew rate in mA/sec
   END_VAR
   VAR_IN_OUT
      RealValue : Real;
   END_VAR
   VAR
      Slew : Bool;
      Inc_TON : TON_TIME;
   END_VAR
   VAR_TEMP
      tempReal : Real;
   END_VAR
BEGIN

REGION Network 1: Slew rate in mA/sec
   // Increase the input value by the slew rate
   // Increasing every 10ms divide rate by 100
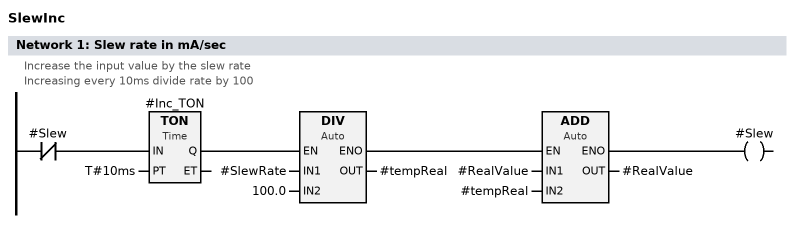
   RUNG wire#powerrail
      I_Contact( #Slew )
      { S7_Templates := "time_type := Time" } #Inc_TON.TON(pt := T#10ms, et =>)
      Div(in1 := #SlewRate, in2 := 100.0, out => #tempReal)
      Add(in1 := #RealValue, in2 := #tempReal, out => #RealValue)
      Coil( #Slew )
   END_RUNG
   // the same network as SCL:
   #Inc_TON(IN := NOT #Slew, PT := T#10ms);   // TON
   IF #Inc_TON.Q THEN
       #tempReal := #SlewRate / 100.0;
       #RealValue := #RealValue + #tempReal;
   END_IF;
   #Slew := #Inc_TON.Q;
END_REGION
END_FUNCTION_BLOCK

FUNCTION_BLOCK "MU_Spin"   // FB31, LAD
TITLE = MU Spin
{ S7_Optimized_Access := 'TRUE' }
// Written BY Kristopher Gimenez Feb 3,2023
// This block is used to control the TD MU Spin mode
// stored: AutoNumber false, MemoryReserve 100, SetENOAutomatically false
   VAR_OUTPUT
      FlowFwdmAOut : Real;
      TorqmAOut : Real;
      FwdEnableP1 : Bool;
      FwdEnableP2 : Bool;
      TorqEn : Bool;
   END_VAR
   VAR
      LinkExtSw_Last : Bool;
      LinkRetSw_Last : Bool;
      MUSpinComplete : Bool;
   END_VAR
   VAR_TEMP
      TorqPSITemp : Real;
   END_VAR
   VAR_TEMP   // added for the SCL form of the ladder/FBD networks
      _w1 : Bool;
      _w2 : Bool;
      _w3 : Bool;
   END_VAR
BEGIN

REGION Network 1: Speed Adjust
   // If PTO confirmed in MU Spin mode allow user to adjust spin speed setpoint using Link Tilt Joysticks
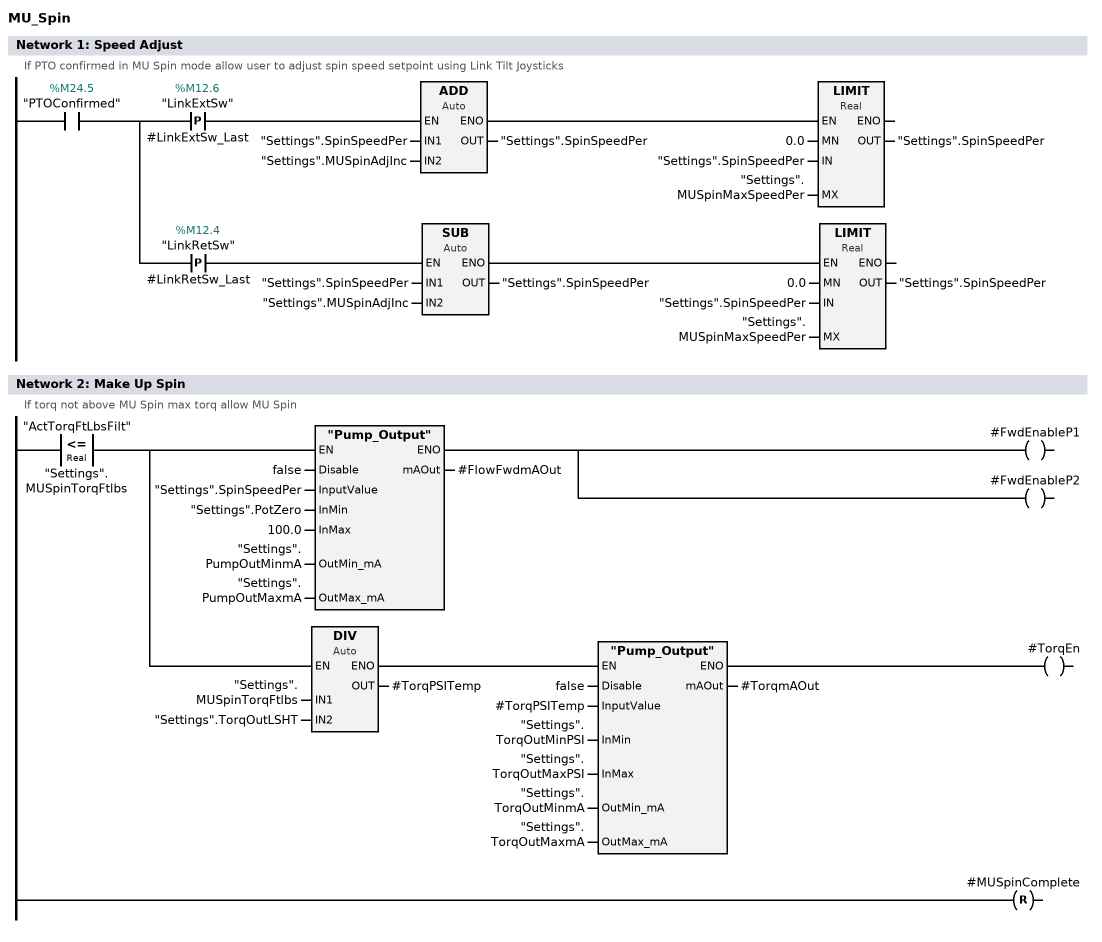
   RUNG wire#powerrail
      Contact( "PTOConfirmed" )
      wire#w1
      P_Contact(operand := "LinkExtSw", bit := #LinkExtSw_Last)
      Add(in1 := "Settings".SpinSpeedPer, in2 := "Settings".MUSpinAdjInc, out => "Settings".SpinSpeedPer)
      { S7_Templates := "value_type := Real" } Limit(mn := 0.0, in := "Settings".SpinSpeedPer, mx := "Settings".MUSpinMaxSpeedPer, out => "Settings".SpinSpeedPer)
   END_RUNG
   RUNG wire#w1
      P_Contact(operand := "LinkRetSw", bit := #LinkRetSw_Last)
      Sub(in1 := "Settings".SpinSpeedPer, in2 := "Settings".MUSpinAdjInc, out => "Settings".SpinSpeedPer)
      { S7_Templates := "value_type := Real" } Limit(mn := 0.0, in := "Settings".SpinSpeedPer, mx := "Settings".MUSpinMaxSpeedPer, out => "Settings".SpinSpeedPer)
   END_RUNG
   // the same network as SCL:
   #_w1 := "PTOConfirmed" AND "LinkExtSw" AND NOT #LinkExtSw_Last;   // rising edge of "LinkExtSw"
   #LinkExtSw_Last := "LinkExtSw";
   IF #_w1 THEN
       "Settings".SpinSpeedPer := "Settings".SpinSpeedPer + "Settings".MUSpinAdjInc;
       "Settings".SpinSpeedPer := LIMIT(MN := 0.0, IN := "Settings".SpinSpeedPer, MX := "Settings".MUSpinMaxSpeedPer);
   END_IF;
   #_w2 := "PTOConfirmed" AND "LinkRetSw" AND NOT #LinkRetSw_Last;   // rising edge of "LinkRetSw"
   #LinkRetSw_Last := "LinkRetSw";
   IF #_w2 THEN
       "Settings".SpinSpeedPer := "Settings".SpinSpeedPer - "Settings".MUSpinAdjInc;
       "Settings".SpinSpeedPer := LIMIT(MN := 0.0, IN := "Settings".SpinSpeedPer, MX := "Settings".MUSpinMaxSpeedPer);
   END_IF;
END_REGION

REGION Network 2: Make Up Spin
   // If torq not above MU Spin max torq allow MU Spin
   RUNG wire#powerrail
      { S7_Templates := "SrcType := Real" } LE_Contact(in1 := "ActTorqFtLbsFilt", in2 := "Settings".MUSpinTorqFtlbs)
      wire#w1
      "Pump_Output"(Disable := false, InputValue := "Settings".SpinSpeedPer, InMin := "Settings".PotZero, InMax := 100.0, OutMin_mA := "Settings".PumpOutMinmA, OutMax_mA := "Settings".PumpOutMaxmA, mAOut => #FlowFwdmAOut)
      wire#w2
      Coil( #FwdEnableP1 )
   END_RUNG
   RUNG wire#w2
      Coil( #FwdEnableP2 )
   END_RUNG
   RUNG wire#w1
      Div(in1 := "Settings".MUSpinTorqFtlbs, in2 := "Settings".TorqOutLSHT, out => #TorqPSITemp)
      "Pump_Output"(Disable := false, InputValue := #TorqPSITemp, InMin := "Settings".TorqOutMinPSI, InMax := "Settings".TorqOutMaxPSI, OutMin_mA := "Settings".TorqOutMinmA, OutMax_mA := "Settings".TorqOutMaxmA, mAOut => #TorqmAOut)
      Coil( #TorqEn )
   END_RUNG
   RUNG wire#powerrail
      R_Coil( #MUSpinComplete )
   END_RUNG
   // the same network as SCL:
   #_w2 := "ActTorqFtLbsFilt" <= "Settings".MUSpinTorqFtlbs;
   "Pump_Output"(EN := "ActTorqFtLbsFilt" <= "Settings".MUSpinTorqFtlbs,
                 Disable := false,
                 InputValue := "Settings".SpinSpeedPer,
                 InMin := "Settings".PotZero,
                 InMax := 100.0,
                 OutMin_mA := "Settings".PumpOutMinmA,
                 OutMax_mA := "Settings".PumpOutMaxmA,
                 mAOut => #FlowFwdmAOut,
                 ENO => #_w1);
   #FwdEnableP1 := #_w1;
   #FwdEnableP2 := #_w1;
   IF #_w2 THEN #TorqPSITemp := "Settings".MUSpinTorqFtlbs / "Settings".TorqOutLSHT; END_IF;
   "Pump_Output"(EN := #_w2,
                 Disable := false,
                 InputValue := #TorqPSITemp,
                 InMin := "Settings".TorqOutMinPSI,
                 InMax := "Settings".TorqOutMaxPSI,
                 OutMin_mA := "Settings".TorqOutMinmA,
                 OutMax_mA := "Settings".TorqOutMaxmA,
                 mAOut => #TorqmAOut,
                 ENO => #_w3);
   #TorqEn := #_w3;
   #MUSpinComplete := FALSE;
END_REGION
END_FUNCTION_BLOCK

FUNCTION_BLOCK "MU_Torq"   // FB32, LAD
TITLE = MU Torq
{ S7_Optimized_Access := 'TRUE' }
// Written BY Kristopher Gimenez Feb 3,2023
// This block is used to control the TD MU Torq mode
// stored: AutoNumber false, MemoryReserve 100, SetENOAutomatically false
   VAR_INPUT
      Start : Bool;
   END_VAR
   VAR_OUTPUT
      FlowFwdmAOut : Real;
      TorqmAOut : Real;
      EnableP1 : Bool;
      EnableP2 { ExternalWritable := 'False'} : Bool;
      TorqEn : Bool;
      MUSeqRunning : Bool;
   END_VAR
   VAR
      MUspeed : Real;
      PumpToggle : Bool;   // Bit will toggle each make up sequence to choose which pump to stroke. 0 = P1, 1 = P2
      AutoMUComplete : Bool;
      RampDown : Bool;   // Bit to know system need to ramp down
      RampDownComplete : Bool;   // Indicates Ramp Down completed
      MUComplete_TON { S7_SetPoint := 'True'} : TON_TIME;
      TorqUserSetmA : Real;
      AutoMUInc_TON { S7_SetPoint := 'True'} : TON_TIME;
      Torq_Ramp { S7_SetPoint := 'True'} : RampFunction;
      Flow_Ramp { S7_SetPoint := 'True'} : RampFunction;
      TorqRampInmA { S7_SetPoint := 'True'} : Real;   // Value assigned to ramp fucntion to get ramped output
      FlowRampInmA : Real;   // Value assigned to ramp fucntion to get ramped ouput
      MUSeqRunLast : Bool;
   END_VAR
   VAR_TEMP
      TorqPSITemp : Real;
      tempReal : Real;
      toggleTemp : Bool;
   END_VAR
   VAR_TEMP   // added for the SCL form of the ladder/FBD networks
      _w1 : Bool;
      _w2 : Bool;
      _w3 : Bool;
      _w4 : Bool;
      _w5 : Bool;
      _w6 : Bool;
      _w7 : Bool;
   END_VAR
BEGIN

REGION Network 1: Set Running
   // Set running bit and trigger resets when starting a MU sequence
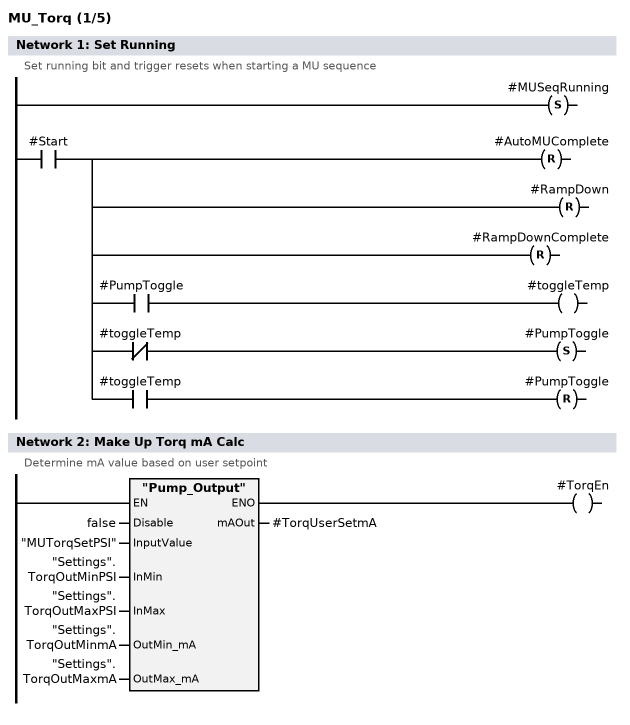
   RUNG wire#powerrail
      S_Coil( #MUSeqRunning )
   END_RUNG
   RUNG wire#powerrail
      Contact( #Start )
      wire#w1
      R_Coil( #AutoMUComplete )
   END_RUNG
   RUNG wire#w1
      R_Coil( #RampDown )
   END_RUNG
   RUNG wire#w1
      R_Coil( #RampDownComplete )
   END_RUNG
   RUNG wire#w1
      Contact( #PumpToggle )
      Coil( #toggleTemp )
   END_RUNG
   RUNG wire#w1
      I_Contact( #toggleTemp )
      S_Coil( #PumpToggle )
   END_RUNG
   RUNG wire#w1
      Contact( #toggleTemp )
      R_Coil( #PumpToggle )
   END_RUNG
   // the same network as SCL:
   #MUSeqRunning := TRUE;
   IF #Start THEN
       #AutoMUComplete := FALSE;
       #RampDown := FALSE;
       #RampDownComplete := FALSE;
   END_IF;
   #toggleTemp := #Start AND #PumpToggle;
   IF #Start AND NOT #toggleTemp THEN #PumpToggle := TRUE; END_IF;
   IF #Start AND #toggleTemp THEN #PumpToggle := FALSE; END_IF;
END_REGION

REGION Network 2: Make Up Torq mA Calc
   // Determine mA value based on user setpoint
   RUNG wire#powerrail
      "Pump_Output"(Disable := false, InputValue := "MUTorqSetPSI", InMin := "Settings".TorqOutMinPSI, InMax := "Settings".TorqOutMaxPSI, OutMin_mA := "Settings".TorqOutMinmA, OutMax_mA := "Settings".TorqOutMaxmA, mAOut => #TorqUserSetmA)
      Coil( #TorqEn )
   END_RUNG
   // the same network as SCL:
   "Pump_Output"(Disable := false,
                 InputValue := "MUTorqSetPSI",
                 InMin := "Settings".TorqOutMinPSI,
                 InMax := "Settings".TorqOutMaxPSI,
                 OutMin_mA := "Settings".TorqOutMinmA,
                 OutMax_mA := "Settings".TorqOutMaxmA,
                 mAOut => #TorqUserSetmA,
                 ENO => #_w1);
   #TorqEn := #_w1;
END_REGION

REGION Network 3: Mu torque speed setting based on torque setpoint
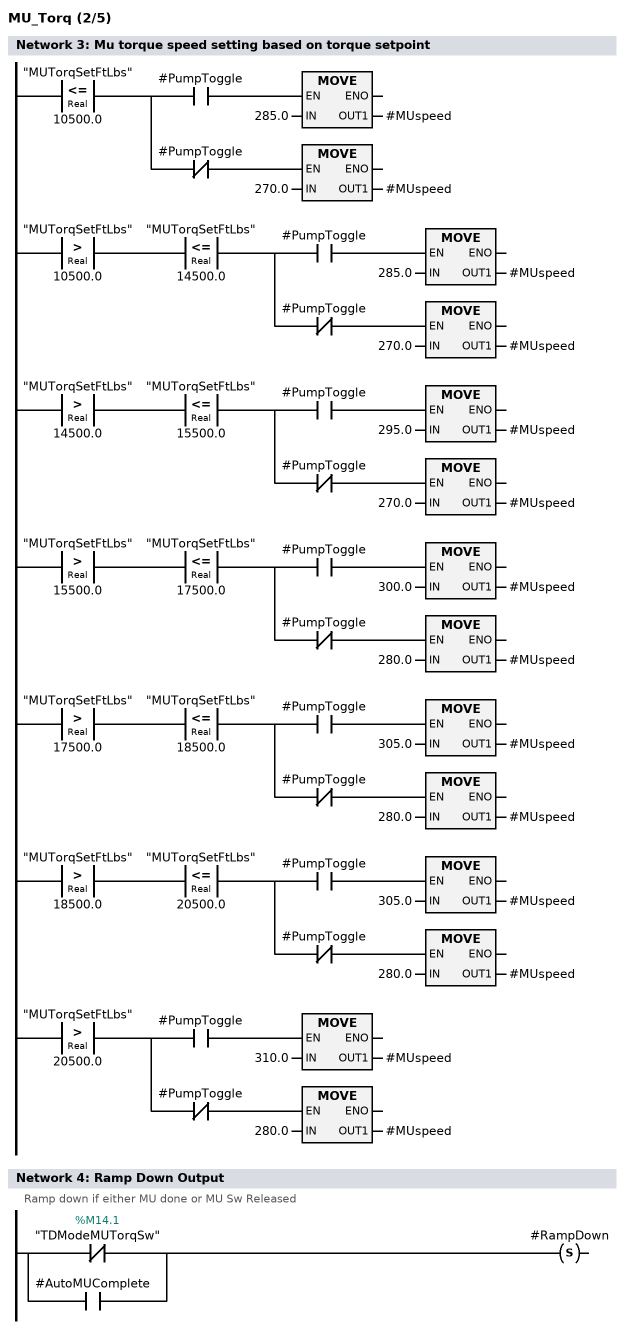
   RUNG wire#powerrail
      { S7_Templates := "SrcType := Real" } LE_Contact(in1 := "MUTorqSetFtLbs", in2 := 10500.0)
      wire#w1
      Contact( #PumpToggle )
      Move(in := 285.0, out1 => #MUspeed)
   END_RUNG
   RUNG wire#w1
      I_Contact( #PumpToggle )
      Move(in := 270.0, out1 => #MUspeed)
   END_RUNG
   RUNG wire#powerrail
      { S7_Templates := "SrcType := Real" } GT_Contact(in1 := "MUTorqSetFtLbs", in2 := 10500.0)
      { S7_Templates := "SrcType := Real" } LE_Contact(in1 := "MUTorqSetFtLbs", in2 := 14500.0)
      wire#w2
      Contact( #PumpToggle )
      Move(in := 285.0, out1 => #MUspeed)
   END_RUNG
   RUNG wire#w2
      I_Contact( #PumpToggle )
      Move(in := 270.0, out1 => #MUspeed)
   END_RUNG
   RUNG wire#powerrail
      { S7_Templates := "SrcType := Real" } GT_Contact(in1 := "MUTorqSetFtLbs", in2 := 14500.0)
      { S7_Templates := "SrcType := Real" } LE_Contact(in1 := "MUTorqSetFtLbs", in2 := 15500.0)
      wire#w3
      Contact( #PumpToggle )
      Move(in := 295.0, out1 => #MUspeed)
   END_RUNG
   RUNG wire#w3
      I_Contact( #PumpToggle )
      Move(in := 270.0, out1 => #MUspeed)
   END_RUNG
   RUNG wire#powerrail
      { S7_Templates := "SrcType := Real" } GT_Contact(in1 := "MUTorqSetFtLbs", in2 := 15500.0)
      { S7_Templates := "SrcType := Real" } LE_Contact(in1 := "MUTorqSetFtLbs", in2 := 17500.0)
      wire#w4
      Contact( #PumpToggle )
      Move(in := 300.0, out1 => #MUspeed)
   END_RUNG
   RUNG wire#w4
      I_Contact( #PumpToggle )
      Move(in := 280.0, out1 => #MUspeed)
   END_RUNG
   RUNG wire#powerrail
      { S7_Templates := "SrcType := Real" } GT_Contact(in1 := "MUTorqSetFtLbs", in2 := 17500.0)
      { S7_Templates := "SrcType := Real" } LE_Contact(in1 := "MUTorqSetFtLbs", in2 := 18500.0)
      wire#w5
      Contact( #PumpToggle )
      Move(in := 305.0, out1 => #MUspeed)
   END_RUNG
   RUNG wire#w5
      I_Contact( #PumpToggle )
      Move(in := 280.0, out1 => #MUspeed)
   END_RUNG
   RUNG wire#powerrail
      { S7_Templates := "SrcType := Real" } GT_Contact(in1 := "MUTorqSetFtLbs", in2 := 18500.0)
      { S7_Templates := "SrcType := Real" } LE_Contact(in1 := "MUTorqSetFtLbs", in2 := 20500.0)
      wire#w6
      Contact( #PumpToggle )
      Move(in := 305.0, out1 => #MUspeed)
   END_RUNG
   RUNG wire#w6
      I_Contact( #PumpToggle )
      Move(in := 280.0, out1 => #MUspeed)
   END_RUNG
   RUNG wire#powerrail
      { S7_Templates := "SrcType := Real" } GT_Contact(in1 := "MUTorqSetFtLbs", in2 := 20500.0)
      wire#w7
      Contact( #PumpToggle )
      Move(in := 310.0, out1 => #MUspeed)
   END_RUNG
   RUNG wire#w7
      I_Contact( #PumpToggle )
      Move(in := 280.0, out1 => #MUspeed)
   END_RUNG
   // the same network as SCL:
   #_w1 := "MUTorqSetFtLbs" <= 10500.0;
   IF #_w1 AND #PumpToggle THEN #MUspeed := 285.0; END_IF;
   IF #_w1 AND NOT #PumpToggle THEN #MUspeed := 270.0; END_IF;
   #_w2 := ("MUTorqSetFtLbs" > 10500.0) AND ("MUTorqSetFtLbs" <= 14500.0);
   IF #_w2 AND #PumpToggle THEN #MUspeed := 285.0; END_IF;
   IF #_w2 AND NOT #PumpToggle THEN #MUspeed := 270.0; END_IF;
   #_w3 := ("MUTorqSetFtLbs" > 14500.0) AND ("MUTorqSetFtLbs" <= 15500.0);
   IF #_w3 AND #PumpToggle THEN #MUspeed := 295.0; END_IF;
   IF #_w3 AND NOT #PumpToggle THEN #MUspeed := 270.0; END_IF;
   #_w4 := ("MUTorqSetFtLbs" > 15500.0) AND ("MUTorqSetFtLbs" <= 17500.0);
   IF #_w4 AND #PumpToggle THEN #MUspeed := 300.0; END_IF;
   IF #_w4 AND NOT #PumpToggle THEN #MUspeed := 280.0; END_IF;
   #_w5 := ("MUTorqSetFtLbs" > 17500.0) AND ("MUTorqSetFtLbs" <= 18500.0);
   IF #_w5 AND #PumpToggle THEN #MUspeed := 305.0; END_IF;
   IF #_w5 AND NOT #PumpToggle THEN #MUspeed := 280.0; END_IF;
   #_w6 := ("MUTorqSetFtLbs" > 18500.0) AND ("MUTorqSetFtLbs" <= 20500.0);
   IF #_w6 AND #PumpToggle THEN #MUspeed := 305.0; END_IF;
   IF #_w6 AND NOT #PumpToggle THEN #MUspeed := 280.0; END_IF;
   #_w7 := "MUTorqSetFtLbs" > 20500.0;
   IF #_w7 AND #PumpToggle THEN #MUspeed := 310.0; END_IF;
   IF #_w7 AND NOT #PumpToggle THEN #MUspeed := 280.0; END_IF;
END_REGION

REGION Network 4: Ramp Down Output
   // Ramp down if either MU done or MU Sw Released
   RUNG wire#powerrail
      I_Contact( "TDModeMUTorqSw" )
      wire#w1
      S_Coil( #RampDown )
   END_RUNG
   RUNG wire#powerrail
      Contact( #AutoMUComplete )
   END_RUNG wire#w1
   // the same network as SCL:
   IF NOT "TDModeMUTorqSw" OR #AutoMUComplete THEN #RampDown := TRUE; END_IF;
END_REGION

REGION Network 5: Assign Torq Ramp Parameters
   // Set Torq Ramp settings as needed. If Transducer faulted use default values. If no TX fault, in Auto Mode set value based on Torq feedback
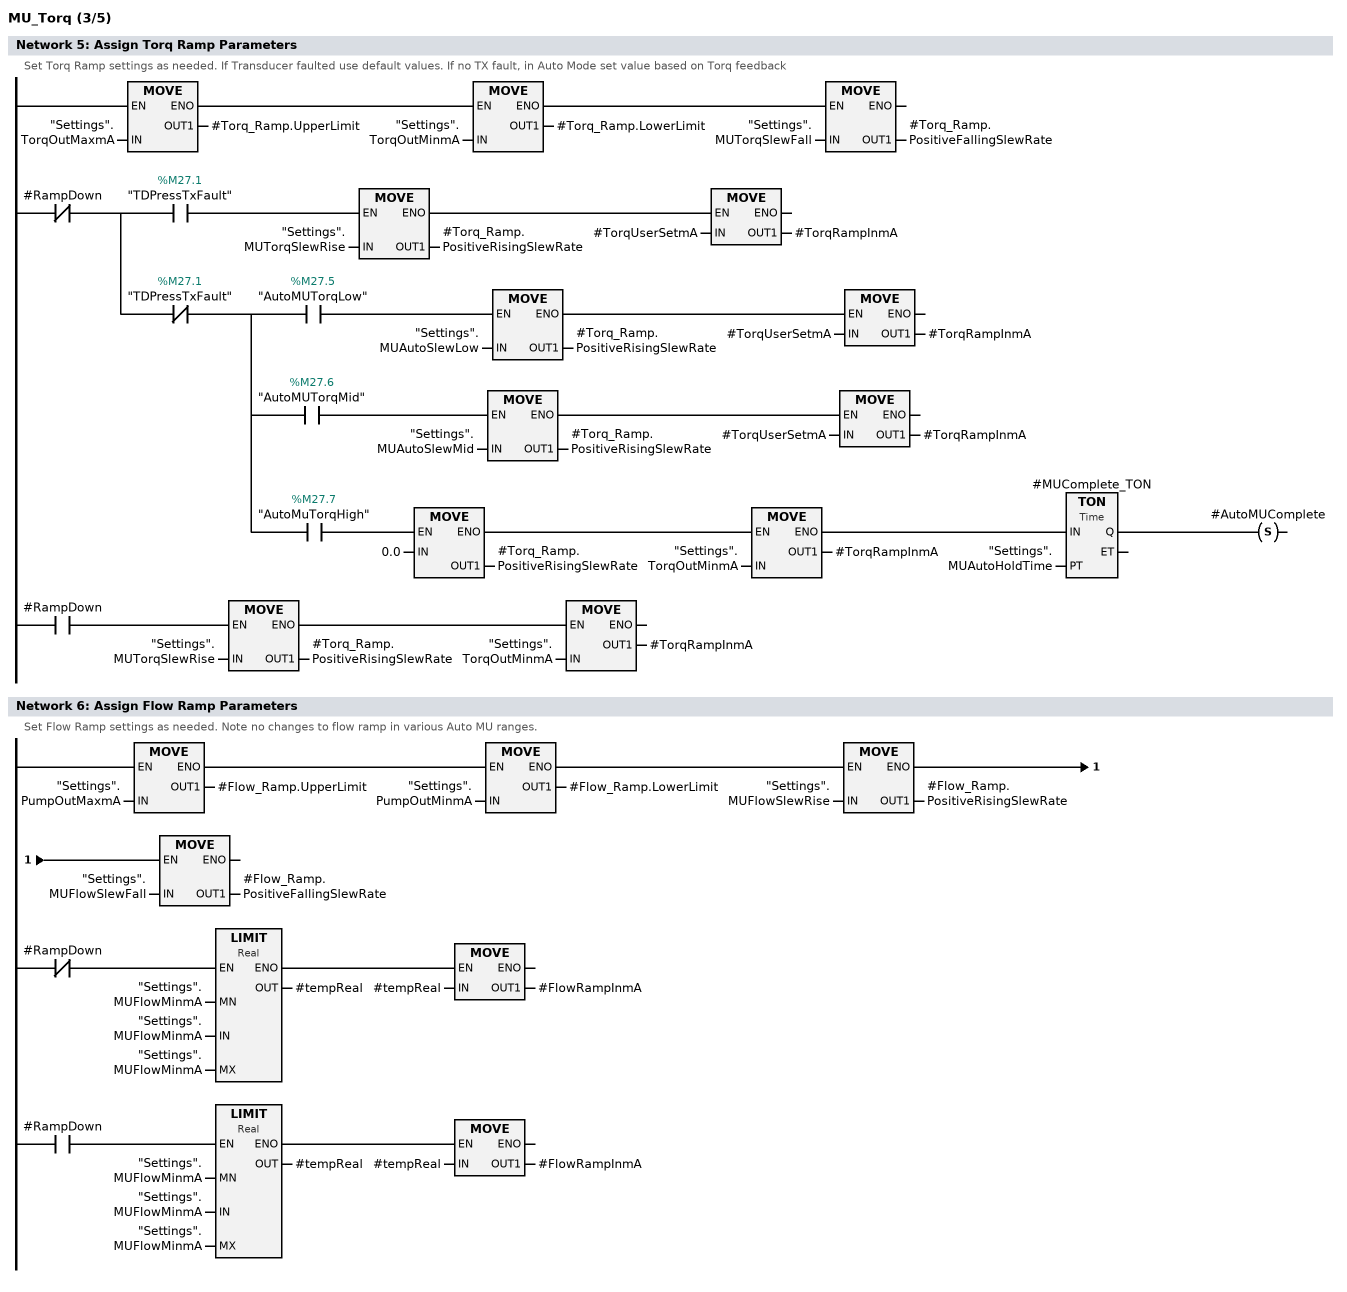
   RUNG wire#powerrail
      Move(in := "Settings".TorqOutMaxmA, out1 => #Torq_Ramp.UpperLimit)
      Move(in := "Settings".TorqOutMinmA, out1 => #Torq_Ramp.LowerLimit)
      Move(in := "Settings".MUTorqSlewFall, out1 => #Torq_Ramp.PositiveFallingSlewRate)
   END_RUNG
   RUNG wire#powerrail
      I_Contact( #RampDown )
      wire#w1
      Contact( "TDPressTxFault" )
      Move(in := "Settings".MUTorqSlewRise, out1 => #Torq_Ramp.PositiveRisingSlewRate)
      Move(in := #TorqUserSetmA, out1 => #TorqRampInmA)
   END_RUNG
   RUNG wire#w1
      I_Contact( "TDPressTxFault" )
      wire#w2
      Contact( "AutoMUTorqLow" )
      Move(in := "Settings".MUAutoSlewLow, out1 => #Torq_Ramp.PositiveRisingSlewRate)
      Move(in := #TorqUserSetmA, out1 => #TorqRampInmA)
   END_RUNG
   RUNG wire#w2
      Contact( "AutoMUTorqMid" )
      Move(in := "Settings".MUAutoSlewMid, out1 => #Torq_Ramp.PositiveRisingSlewRate)
      Move(in := #TorqUserSetmA, out1 => #TorqRampInmA)
   END_RUNG
   RUNG wire#w2
      Contact( "AutoMuTorqHigh" )
      Move(in := 0.0, out1 => #Torq_Ramp.PositiveRisingSlewRate)
      Move(in := "Settings".TorqOutMinmA, out1 => #TorqRampInmA)
      { S7_Templates := "time_type := Time" } #MUComplete_TON.TON(pt := "Settings".MUAutoHoldTime, et =>)
      S_Coil( #AutoMUComplete )
   END_RUNG
   RUNG wire#powerrail
      Contact( #RampDown )
      Move(in := "Settings".MUTorqSlewRise, out1 => #Torq_Ramp.PositiveRisingSlewRate)
      Move(in := "Settings".TorqOutMinmA, out1 => #TorqRampInmA)
   END_RUNG
   // the same network as SCL:
   #Torq_Ramp.UpperLimit := "Settings".TorqOutMaxmA;
   #Torq_Ramp.LowerLimit := "Settings".TorqOutMinmA;
   #Torq_Ramp.PositiveFallingSlewRate := "Settings".MUTorqSlewFall;
   IF NOT #RampDown AND "TDPressTxFault" THEN
       #Torq_Ramp.PositiveRisingSlewRate := "Settings".MUTorqSlewRise;
       #TorqRampInmA := #TorqUserSetmA;
   END_IF;
   #_w1 := NOT #RampDown AND NOT "TDPressTxFault";
   IF #_w1 AND "AutoMUTorqLow" THEN
       #Torq_Ramp.PositiveRisingSlewRate := "Settings".MUAutoSlewLow;
       #TorqRampInmA := #TorqUserSetmA;
   END_IF;
   IF #_w1 AND "AutoMUTorqMid" THEN
       #Torq_Ramp.PositiveRisingSlewRate := "Settings".MUAutoSlewMid;
       #TorqRampInmA := #TorqUserSetmA;
   END_IF;
   #_w2 := #_w1 AND "AutoMuTorqHigh";
   IF #_w2 THEN
       #Torq_Ramp.PositiveRisingSlewRate := 0.0;
       #TorqRampInmA := "Settings".TorqOutMinmA;
   END_IF;
   #MUComplete_TON(IN := #_w2, PT := "Settings".MUAutoHoldTime);   // TON
   IF #MUComplete_TON.Q THEN #AutoMUComplete := TRUE; END_IF;
   IF #RampDown THEN
       #Torq_Ramp.PositiveRisingSlewRate := "Settings".MUTorqSlewRise;
       #TorqRampInmA := "Settings".TorqOutMinmA;
   END_IF;
END_REGION

REGION Network 6: Assign Flow Ramp Parameters
   // Set Flow Ramp settings as needed. Note no changes to flow ramp in various Auto MU ranges.
   RUNG wire#powerrail
      Move(in := "Settings".PumpOutMaxmA, out1 => #Flow_Ramp.UpperLimit)
      Move(in := "Settings".PumpOutMinmA, out1 => #Flow_Ramp.LowerLimit)
      Move(in := "Settings".MUFlowSlewRise, out1 => #Flow_Ramp.PositiveRisingSlewRate)
      Move(in := "Settings".MUFlowSlewFall, out1 => #Flow_Ramp.PositiveFallingSlewRate)
   END_RUNG
   RUNG wire#powerrail
      I_Contact( #RampDown )
      { S7_Templates := "value_type := Real" } Limit(mn := "Settings".MUFlowMinmA, in := "Settings".MUFlowMinmA, mx := "Settings".MUFlowMinmA, out => #tempReal)
      Move(in := #tempReal, out1 => #FlowRampInmA)
   END_RUNG
   RUNG wire#powerrail
      Contact( #RampDown )
      { S7_Templates := "value_type := Real" } Limit(mn := "Settings".MUFlowMinmA, in := "Settings".MUFlowMinmA, mx := "Settings".MUFlowMinmA, out => #tempReal)
      Move(in := #tempReal, out1 => #FlowRampInmA)
   END_RUNG
   // the same network as SCL:
   #Flow_Ramp.UpperLimit := "Settings".PumpOutMaxmA;
   #Flow_Ramp.LowerLimit := "Settings".PumpOutMinmA;
   #Flow_Ramp.PositiveRisingSlewRate := "Settings".MUFlowSlewRise;
   #Flow_Ramp.PositiveFallingSlewRate := "Settings".MUFlowSlewFall;
   IF NOT #RampDown THEN
       #tempReal := LIMIT(MN := "Settings".MUFlowMinmA, IN := "Settings".MUFlowMinmA, MX := "Settings".MUFlowMinmA);
       #FlowRampInmA := #tempReal;
   END_IF;
   IF #RampDown THEN
       #tempReal := LIMIT(MN := "Settings".MUFlowMinmA, IN := "Settings".MUFlowMinmA, MX := "Settings".MUFlowMinmA);
       #FlowRampInmA := #tempReal;
   END_IF;
END_REGION

REGION Network 7: Ramp mA Signals
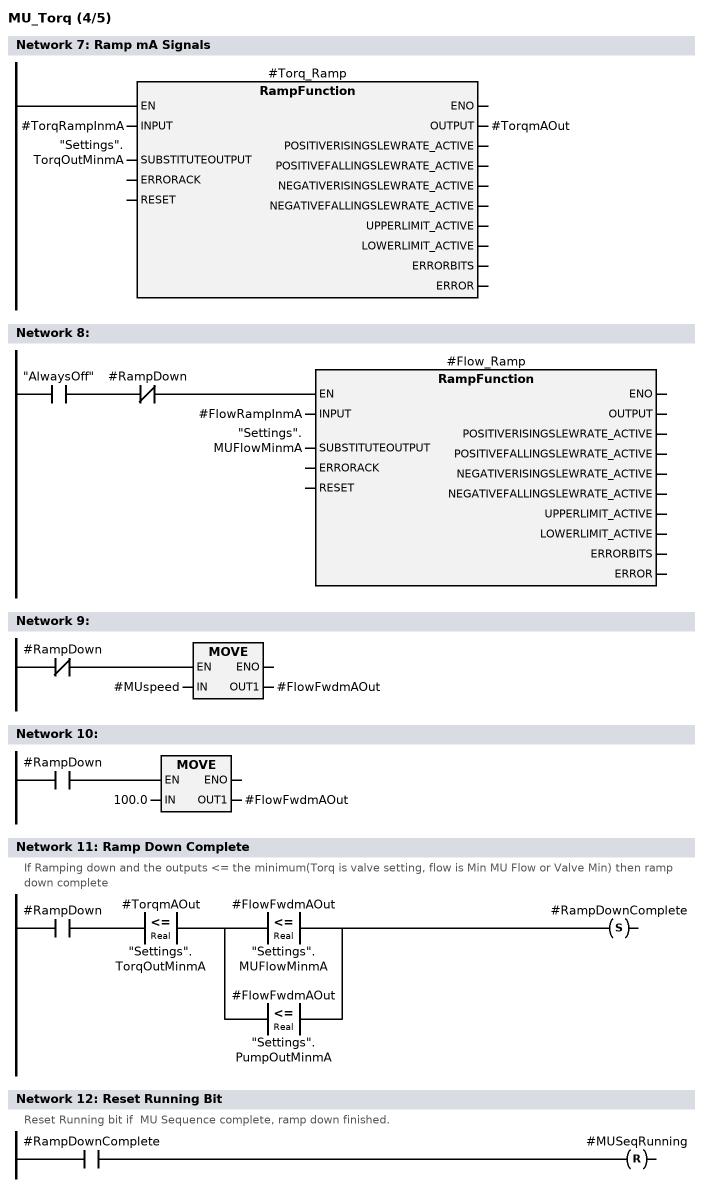
   RUNG wire#powerrail
      #Torq_Ramp.RampFunction(Input := #TorqRampInmA, SubstituteOutput := "Settings".TorqOutMinmA, ErrorAck :=, Reset :=, Output => #TorqmAOut, PositiveRisingSlewRate_Active =>, PositiveFallingSlewRate_Active =>, NegativeRisingSlewRate_Active =>, NegativeFallingSlewRate_Active =>, UpperLimit_Active =>, LowerLimit_Active =>, ErrorBits =>, Error =>)
   END_RUNG
   // the same network as SCL:
   #Torq_Ramp(Input := #TorqRampInmA, SubstituteOutput := "Settings".TorqOutMinmA, Output => #TorqmAOut);   // RampFunction
END_REGION

REGION Network 8
   RUNG wire#powerrail
      Contact( "AlwaysOff" )
      I_Contact( #RampDown )
      #Flow_Ramp.RampFunction(Input := #FlowRampInmA, SubstituteOutput := "Settings".MUFlowMinmA, ErrorAck :=, Reset :=, Output =>, PositiveRisingSlewRate_Active =>, PositiveFallingSlewRate_Active =>, NegativeRisingSlewRate_Active =>, NegativeFallingSlewRate_Active =>, UpperLimit_Active =>, LowerLimit_Active =>, ErrorBits =>, Error =>)
   END_RUNG
   // the same network as SCL:
   IF "AlwaysOff" AND NOT #RampDown THEN
       #Flow_Ramp(Input := #FlowRampInmA, SubstituteOutput := "Settings".MUFlowMinmA);   // RampFunction
   END_IF;
END_REGION

REGION Network 9
   RUNG wire#powerrail
      I_Contact( #RampDown )
      Move(in := #MUspeed, out1 => #FlowFwdmAOut)
   END_RUNG
   // the same network as SCL:
   IF NOT #RampDown THEN #FlowFwdmAOut := #MUspeed; END_IF;
END_REGION

REGION Network 10
   RUNG wire#powerrail
      Contact( #RampDown )
      Move(in := 100.0, out1 => #FlowFwdmAOut)
   END_RUNG
   // the same network as SCL:
   IF #RampDown THEN #FlowFwdmAOut := 100.0; END_IF;
END_REGION

REGION Network 11: Ramp Down Complete
   // If Ramping down and the outputs <= the minimum(Torq is valve setting, flow is Min MU Flow or Valve Min) then ramp down complete
   RUNG wire#powerrail
      Contact( #RampDown )
      { S7_Templates := "SrcType := Real" } LE_Contact(in1 := #TorqmAOut, in2 := "Settings".TorqOutMinmA)
      wire#w1
      { S7_Templates := "SrcType := Real" } LE_Contact(in1 := #FlowFwdmAOut, in2 := "Settings".MUFlowMinmA)
      wire#w2
      S_Coil( #RampDownComplete )
   END_RUNG
   RUNG wire#w1
      { S7_Templates := "SrcType := Real" } LE_Contact(in1 := #FlowFwdmAOut, in2 := "Settings".PumpOutMinmA)
   END_RUNG wire#w2
   // the same network as SCL:
   IF #RampDown AND (#TorqmAOut <= "Settings".TorqOutMinmA) AND ((#FlowFwdmAOut <= "Settings".MUFlowMinmA) OR (#FlowFwdmAOut <= "Settings".PumpOutMinmA)) THEN
       #RampDownComplete := TRUE;
   END_IF;
END_REGION

REGION Network 12: Reset Running Bit
   // Reset Running bit if  MU Sequence complete, ramp down finished.
   RUNG wire#powerrail
      Contact( #RampDownComplete )
      R_Coil( #MUSeqRunning )
   END_RUNG
   // the same network as SCL:
   IF #RampDownComplete THEN #MUSeqRunning := FALSE; END_IF;
END_REGION

REGION Network 13: Set Outputs
   // Torq always enabled in MU mode. Pumps alternate
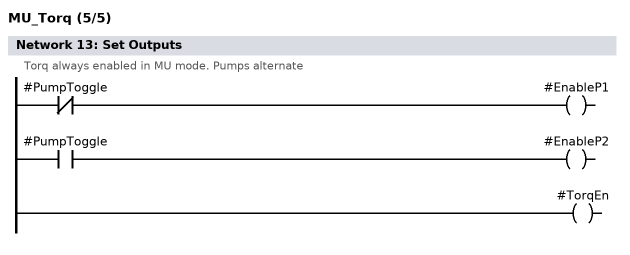
   RUNG wire#powerrail
      I_Contact( #PumpToggle )
      Coil( #EnableP1 )
   END_RUNG
   RUNG wire#powerrail
      Contact( #PumpToggle )
      Coil( #EnableP2 )
   END_RUNG
   RUNG wire#powerrail
      Coil( #TorqEn )
   END_RUNG
   // the same network as SCL:
   #EnableP1 := NOT #PumpToggle;
   #EnableP2 := #PumpToggle;
   #TorqEn := TRUE;
END_REGION
END_FUNCTION_BLOCK

FUNCTION_BLOCK "BO_Torq"   // FB33, LAD
TITLE = Break Out
{ S7_Optimized_Access := 'TRUE' }
// Written BY Kristopher Gimenez Feb 7,2023
// This block is used to control the TD Break Out Torq mode
// stored: AutoNumber false, MemoryReserve 100, SetENOAutomatically false
   VAR_INPUT
      Start : Bool;
   END_VAR
   VAR_OUTPUT
      FlowRevmAOut : Real;
      EnableP1 : Bool;
      EnableP2 { ExternalWritable := 'False'} : Bool;
      BOEn : Bool;
      BOSeqRunning : Bool;
   END_VAR
   VAR
      PumpToggle : Bool;   // Bit will toggle each make up sequence to choose which pump to stroke. 0 = P1, 1 = P2, TBD if using this in BO.
      RampDown : Bool;   // Bit to know system need to ramp down
      RampDownComplete : Bool;   // Indicates Ramp Down completed
      Flow_Ramp { S7_SetPoint := 'True'} : RampFunction;
      FlowRampInmA : Real;   // Value assigned to ramp fucntion to get ramped ouput
      BOFlowmA : Real;
      BOSeqRunLast : Bool;
   END_VAR
   VAR_TEMP
      tempReal : Real;
      toggleTemp : Bool;
   END_VAR
BEGIN

REGION Network 1: Set Running
   // Set running bit and trigger resets when starting a MU sequence
   // Pump Toggle is set but may not be needed for BO mode
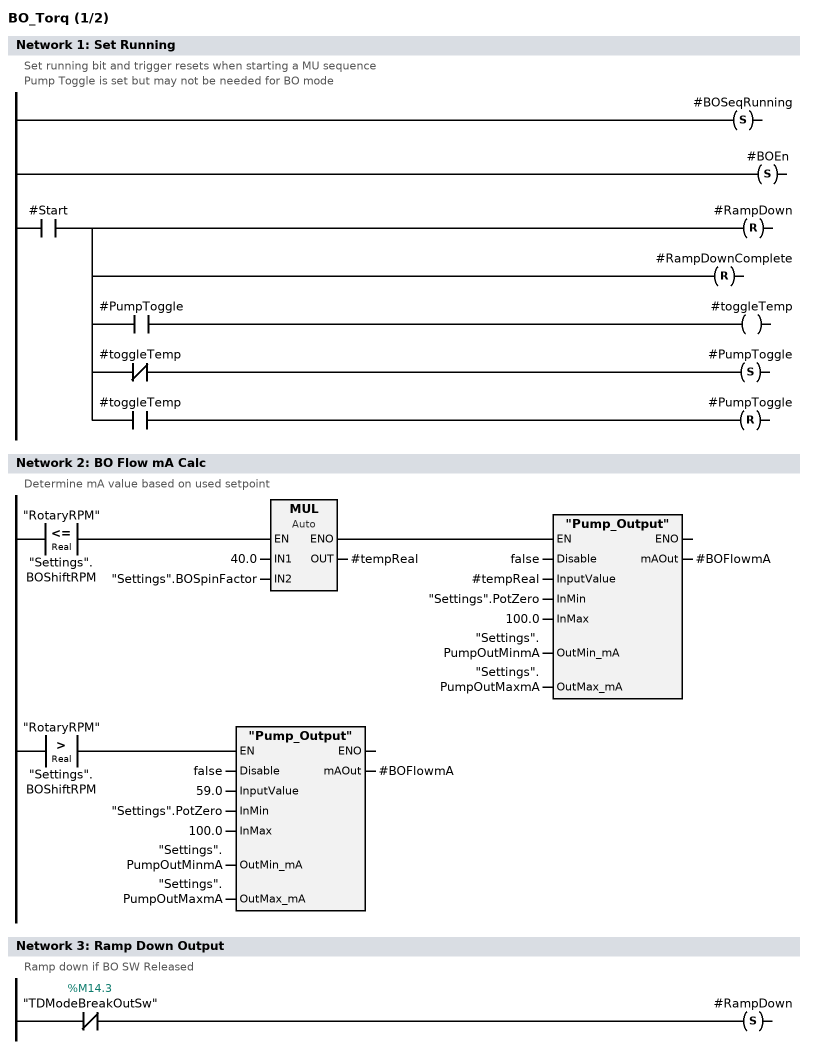
   RUNG wire#powerrail
      S_Coil( #BOSeqRunning )
   END_RUNG
   RUNG wire#powerrail
      S_Coil( #BOEn )
   END_RUNG
   RUNG wire#powerrail
      Contact( #Start )
      wire#w1
      R_Coil( #RampDown )
   END_RUNG
   RUNG wire#w1
      R_Coil( #RampDownComplete )
   END_RUNG
   RUNG wire#w1
      Contact( #PumpToggle )
      Coil( #toggleTemp )
   END_RUNG
   RUNG wire#w1
      I_Contact( #toggleTemp )
      S_Coil( #PumpToggle )
   END_RUNG
   RUNG wire#w1
      Contact( #toggleTemp )
      R_Coil( #PumpToggle )
   END_RUNG
   // the same network as SCL:
   #BOSeqRunning := TRUE;
   #BOEn := TRUE;
   IF #Start THEN
       #RampDown := FALSE;
       #RampDownComplete := FALSE;
   END_IF;
   #toggleTemp := #Start AND #PumpToggle;
   IF #Start AND NOT #toggleTemp THEN #PumpToggle := TRUE; END_IF;
   IF #Start AND #toggleTemp THEN #PumpToggle := FALSE; END_IF;
END_REGION

REGION Network 2: BO Flow mA Calc
   // Determine mA value based on used setpoint
   RUNG wire#powerrail
      { S7_Templates := "SrcType := Real" } LE_Contact(in1 := "RotaryRPM", in2 := "Settings".BOShiftRPM)
      Mul(in1 := 40.0, in2 := "Settings".BOSpinFactor, out => #tempReal)
      "Pump_Output"(Disable := false, InputValue := #tempReal, InMin := "Settings".PotZero, InMax := 100.0, OutMin_mA := "Settings".PumpOutMinmA, OutMax_mA := "Settings".PumpOutMaxmA, mAOut => #BOFlowmA)
   END_RUNG
   RUNG wire#powerrail
      { S7_Templates := "SrcType := Real" } GT_Contact(in1 := "RotaryRPM", in2 := "Settings".BOShiftRPM)
      "Pump_Output"(Disable := false, InputValue := 59.0, InMin := "Settings".PotZero, InMax := 100.0, OutMin_mA := "Settings".PumpOutMinmA, OutMax_mA := "Settings".PumpOutMaxmA, mAOut => #BOFlowmA)
   END_RUNG
   // the same network as SCL:
   IF "RotaryRPM" <= "Settings".BOShiftRPM THEN
       #tempReal := 40.0 * "Settings".BOSpinFactor;
       "Pump_Output"(Disable := false,
                     InputValue := #tempReal,
                     InMin := "Settings".PotZero,
                     InMax := 100.0,
                     OutMin_mA := "Settings".PumpOutMinmA,
                     OutMax_mA := "Settings".PumpOutMaxmA,
                     mAOut => #BOFlowmA);
   END_IF;
   IF "RotaryRPM" > "Settings".BOShiftRPM THEN
       "Pump_Output"(Disable := false,
                     InputValue := 59.0,
                     InMin := "Settings".PotZero,
                     InMax := 100.0,
                     OutMin_mA := "Settings".PumpOutMinmA,
                     OutMax_mA := "Settings".PumpOutMaxmA,
                     mAOut => #BOFlowmA);
   END_IF;
END_REGION

REGION Network 3: Ramp Down Output
   // Ramp down if BO SW Released
   RUNG wire#powerrail
      I_Contact( "TDModeBreakOutSw" )
      S_Coil( #RampDown )
   END_RUNG
   // the same network as SCL:
   IF NOT "TDModeBreakOutSw" THEN #RampDown := TRUE; END_IF;
END_REGION

REGION Network 4: Assign Flow Ramp Parameters
   // Set Flow Ramp settings as needed. Note no changes to flow ramp in various Auto MU ranges.
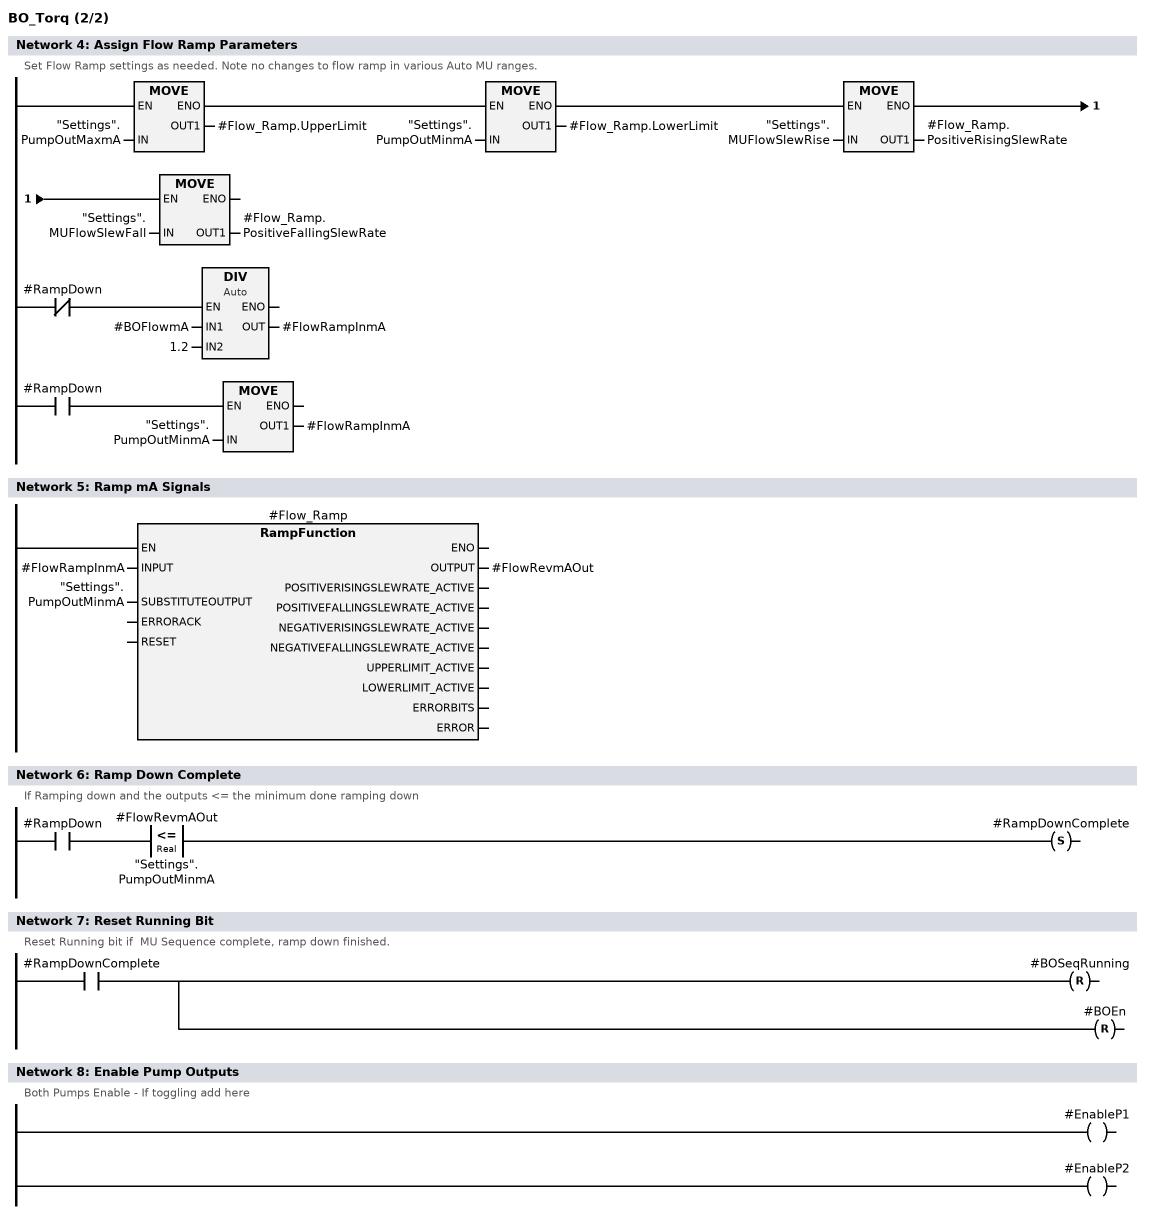
   RUNG wire#powerrail
      Move(in := "Settings".PumpOutMaxmA, out1 => #Flow_Ramp.UpperLimit)
      Move(in := "Settings".PumpOutMinmA, out1 => #Flow_Ramp.LowerLimit)
      Move(in := "Settings".MUFlowSlewRise, out1 => #Flow_Ramp.PositiveRisingSlewRate)
      Move(in := "Settings".MUFlowSlewFall, out1 => #Flow_Ramp.PositiveFallingSlewRate)
   END_RUNG
   RUNG wire#powerrail
      I_Contact( #RampDown )
      Div(in1 := #BOFlowmA, in2 := 1.2, out => #FlowRampInmA)
   END_RUNG
   RUNG wire#powerrail
      Contact( #RampDown )
      Move(in := "Settings".PumpOutMinmA, out1 => #FlowRampInmA)
   END_RUNG
   // the same network as SCL:
   #Flow_Ramp.UpperLimit := "Settings".PumpOutMaxmA;
   #Flow_Ramp.LowerLimit := "Settings".PumpOutMinmA;
   #Flow_Ramp.PositiveRisingSlewRate := "Settings".MUFlowSlewRise;
   #Flow_Ramp.PositiveFallingSlewRate := "Settings".MUFlowSlewFall;
   IF NOT #RampDown THEN #FlowRampInmA := #BOFlowmA / 1.2; END_IF;
   IF #RampDown THEN #FlowRampInmA := "Settings".PumpOutMinmA; END_IF;
END_REGION

REGION Network 5: Ramp mA Signals
   RUNG wire#powerrail
      #Flow_Ramp.RampFunction(Input := #FlowRampInmA, SubstituteOutput := "Settings".PumpOutMinmA, ErrorAck :=, Reset :=, Output => #FlowRevmAOut, PositiveRisingSlewRate_Active =>, PositiveFallingSlewRate_Active =>, NegativeRisingSlewRate_Active =>, NegativeFallingSlewRate_Active =>, UpperLimit_Active =>, LowerLimit_Active =>, ErrorBits =>, Error =>)
   END_RUNG
   // the same network as SCL:
   #Flow_Ramp(Input := #FlowRampInmA, SubstituteOutput := "Settings".PumpOutMinmA, Output => #FlowRevmAOut);   // RampFunction
END_REGION

REGION Network 6: Ramp Down Complete
   // If Ramping down and the outputs <= the minimum done ramping down
   RUNG wire#powerrail
      Contact( #RampDown )
      { S7_Templates := "SrcType := Real" } LE_Contact(in1 := #FlowRevmAOut, in2 := "Settings".PumpOutMinmA)
      S_Coil( #RampDownComplete )
   END_RUNG
   // the same network as SCL:
   IF #RampDown AND (#FlowRevmAOut <= "Settings".PumpOutMinmA) THEN #RampDownComplete := TRUE; END_IF;
END_REGION

REGION Network 7: Reset Running Bit
   // Reset Running bit if  MU Sequence complete, ramp down finished.
   RUNG wire#powerrail
      Contact( #RampDownComplete )
      wire#w1
      R_Coil( #BOSeqRunning )
   END_RUNG
   RUNG wire#w1
      R_Coil( #BOEn )
   END_RUNG
   // the same network as SCL:
   IF #RampDownComplete THEN
       #BOSeqRunning := FALSE;
       #BOEn := FALSE;
   END_IF;
END_REGION

REGION Network 8: Enable Pump Outputs
   // Both Pumps Enable - If toggling add here
   RUNG wire#powerrail
      Coil( #EnableP1 )
   END_RUNG
   RUNG wire#powerrail
      Coil( #EnableP2 )
   END_RUNG
   // the same network as SCL:
   #EnableP1 := TRUE;
   #EnableP2 := TRUE;
END_REGION
END_FUNCTION_BLOCK

FUNCTION_BLOCK "Oscillate"   // FB34, LAD
TITLE = Oscillator
{ S7_Optimized_Access := 'TRUE' }
// Written BY Kristopher Gimenez Feb 3,2023
// This block is used to control the TD Oscillator
// stored: AutoNumber false, MemoryReserve 100, SetENOAutomatically false
   VAR_INPUT
      Start : Bool;
   END_VAR
   VAR_OUTPUT
      FlowmAOut : Real;
      TorqmAOut : Real;
      EnableP1Fwd : Bool;
      EnableP2Fwd : Bool;
      EnableP1Rev : Bool;
      EnableP2Rev : Bool;
      TorqEn : Bool;
   END_VAR
   VAR
      FlowRev : Bool;   // Set High if flow to be in rev, low if flow fwd
      PumpToggle : Bool;   // Bit will toggle each sequence to choose which pump to stroke. 0 = P1, 1 = P2
      Oscillating : Bool;   // Bit to know oscillator is in Oscillate Mode
      Holding : Bool;   // Bit to know oscillator is in hold mode
      OscState : Int;   // State machine mode
      CalcFlowmA : Real;   // Calculated Output flow mA as adjusted based on control.
      LimitFlowmA : Real;   // Limit mA output if Torq limiting
      HomePosAbsDeg : Real;   // Home position in Absolute Degrees
      HomePosAbsDegNew : Real;
      HomeRelDegNew : Real;
      MinmAHigh : Bool;   // Bit to warn that the Minimum mA setting is too large not allowing to hold
      HoldmALow : Bool;   // Bit to warn that the hold mA setting is too small not allowing to hold
      BumpReactiveTrig : Bool;
      BumpFwdTrig : Bool;
      BumpRevTrig : Bool;
      StartDeg : Real;   // Starting Degree for command
      HoldFwdFastInc { S7_SetPoint := 'True'} : Bool;   // Bit used to slew mA output by increment value
      HoldFwdSlowInc : Bool;   // Bit used to slew mA output by increment value
      HoldFwdFastIDec : Bool;   // Bit used to slew mA output by decrement value
      HoldFwdSlowDev : Bool;   // Bit used to slew mA output by decrement value
      HoldRevFastInc : Bool;   // Bit used to slew mA output by increment value
      HoldRevSlowInc : Bool;   // Bit used to slew mA output by increment value
      HoldRevFastIDec : Bool;   // Bit used to slew mA output by decrement value
      HoldRevSlowDev : Bool;   // Bit used to slew mA output by decrement value
      HoldFwdTorqLim : Bool;   // Torq limit reached while Bump Fwd during Hold
      HoldRevTorqLim : Bool;   // Torq Limit Reach while Bump Rev Furing Hold
      MinSetWarn_TON { S7_SetPoint := 'True'} : TON_TIME;   // Minimum mA setpoint warning Time On delay
      HoldFWDFast_SlewInc { S7_SetPoint := 'True'} : "SlewInc";
      HoldFWDSlow_SlewInc { S7_SetPoint := 'True'} : "SlewInc";
      HoldFWDSlow_SlewDec { S7_SetPoint := 'True'} : "SlewDec";
      HoldFWDFast_SlewDec { S7_SetPoint := 'True'} : "SlewDec";
      HoldFWDTorqLim_TON { S7_SetPoint := 'True'} : TON_TIME;
      HoldFwdTorqLim_SlewDec { S7_SetPoint := 'True'} : "SlewDec";
      HoldFwdTorqLim_SlewInc { S7_SetPoint := 'True'} : "SlewInc";
      HoldRevTorqLim_TON { S7_SetPoint := 'True'} : TON_TIME;
      HoldRevTorqLimTrig : Bool;
      HoldFwdTorqLimTrig { ExternalAccessible := 'False'; ExternalVisible := 'False'; ExternalWritable := 'False'} : Bool;
      HoldRevTorqLim_SlewDec { S7_SetPoint := 'True'} : "SlewDec";
      HoldRevTorqLim_SlewInc { S7_SetPoint := 'True'} : "SlewInc";
      HoldRevFast_SlewInc { S7_SetPoint := 'True'} : "SlewInc";
      HoldRevSlow_SlewInc { S7_SetPoint := 'True'} : "SlewInc";
      HoldRevSlow_SlewDec { S7_SetPoint := 'True'} : "SlewDec";
      HoldRevFast_SlewDec { S7_SetPoint := 'True'} : "SlewDec";
      OscFwdTorqLim { S7_SetPoint := 'True'} : Bool;   // Torq limit reached while oscillating Fwd
      OscRevTorqLim : Bool;   // Torq Limit Reach while oscillating in Rev
      OscFwdTrig : Bool;   // Trigger bit when starting to move FWD
      OscRevTrig : Bool;   // Trigger bit when starting to move Rev
      HMIBumpFwdLast : Bool;   // Trigger bit holding last state
      HMIBumpRevLast : Bool;   // Trigger bit holding last state
      HMIBumpReactLast : Bool;   // Trigger bit holding last state
      OscFwdAbsDeg : Real;   // Absolute position to be above to finish a fwd oscillation
      OscFwdAbsSlowdown : Real;
      OscRevAbsDeg : Real;   // Absolute position to be below to finish a rev oscillation
      OscRevAbsSlowdown : Real;
      OscFWDTorqLim_TON { S7_SetPoint := 'True'} : TON_TIME;
      OscFwdTorqLimTrig : Bool;
      OscFwdTorqLim_SlewDec { S7_SetPoint := 'True'} : "SlewDec";
      OscFwdTorqLim_SlewInc { S7_SetPoint := 'True'} : "SlewInc";
      OscFWDFast_SlewInc { S7_SetPoint := 'True'} : "SlewInc";
      OscFWDSlow_SlewInc { S7_SetPoint := 'True'} : "SlewInc";
      OscFWDSlow_SlewDec { S7_SetPoint := 'True'} : "SlewDec";
      OscFWDFast_SlewDec { S7_SetPoint := 'True'} : "SlewDec";
      OscRevTorqLim_TON { S7_SetPoint := 'True'} : TON_TIME;
      OscRevTorqLimTrig : Bool;
      OscRevTorqLim_SlewDec { S7_SetPoint := 'True'} : "SlewDec";
      OscRevTorqLim_SlewInc { S7_SetPoint := 'True'} : "SlewInc";
      OscRevFast_SlewInc { S7_SetPoint := 'True'} : "SlewInc";
      OscRevSlow_SlewInc { S7_SetPoint := 'True'} : "SlewInc";
      OscRevSlow_SlewDec { S7_SetPoint := 'True'} : "SlewDec";
      OscRevFast_SlewDec { S7_SetPoint := 'True'} : "SlewDec";
      HomeFwdTrig : Bool;
      HomeFwdTorqLim : Bool;
      HomeFwdTorqLimTrig : Bool;
      HomeFwdTorqLim_SlewDec { S7_SetPoint := 'True'} : "SlewDec";
      HomeFWDTorqLim_TON { S7_SetPoint := 'True'} : TON_TIME;
      HomeFwdTorqLim_SlewInc { S7_SetPoint := 'True'} : "SlewInc";
      HomeFWDFast_SlewInc { S7_SetPoint := 'True'} : "SlewInc";
      HomeFWDSlow_SlewInc { S7_SetPoint := 'True'} : "SlewInc";
      HomeFWDSlow_SlewDec { S7_SetPoint := 'True'} : "SlewDec";
      HomeFWDFast_SlewDec { S7_SetPoint := 'True'} : "SlewDec";
      HomeRevTrig : Bool;
      HomeRevTorqLim_TON { S7_SetPoint := 'True'} : TON_TIME;
      HomeRevTorqLim : Bool;
      HomeRevTorqLimTrig : Bool;
      HomeRevTorqLim_SlewDec { S7_SetPoint := 'True'} : "SlewDec";
      HomeRevTorqLim_SlewInc { S7_SetPoint := 'True'} : "SlewInc";
      HomeRevFast_SlewInc { S7_SetPoint := 'True'} : "SlewInc";
      HomeRevSlow_SlewInc { S7_SetPoint := 'True'} : "SlewInc";
      HomeRevSlow_SlewDec { S7_SetPoint := 'True'} : "SlewDec";
      HomeRevFast_SlewDec { S7_SetPoint := 'True'} : "SlewDec";
      OscHomeLowAbsDeg : Real;   // Abs Home Position minus 1 count range
      OscHomeLow2AbsDeg : Real;   // Abs Home Position minus 2 count range
      OscHomeHighAbsDeg : Real;   // Abs Home Position plus 1 count range
      OscHomeHigh2AbsDeg : Real;   // Abs Home Position plus 2 count range
   END_VAR
   VAR_TEMP
      HomeDegDiff : Real;
      TempSpeedcheck : Bool;
      MaxflowmAOutTemp : Real;
      TorqPSITemp : Real;
      tempReal : Real;
      Bumpfwdptrig : Bool;
      BumpReactptrig : Bool;
      Bumprevptrig : Bool;
      toggleTemp : Bool;   // Bit used to toggle pump toggle bit
   END_VAR
   VAR CONSTANT
      Startup : Int;
      AwaitCmd : Int := 1;   // Osc enabled and stopped. Waiting for user command.
      StartHolding : Int := 100;
      HoldPos : Int := 101;
      HoldBumpFwd : Int := 102;
      HoldBumpRev : Int := 103;
      HoldBumpReactive : Int := 104;
      StartOscillating : Int := 200;
      OscFWD : Int := 201;
      OscRev : Int := 202;
      StopOscillating : Int := 250;
      HomeFwd : Int := 251;
      HomeRev : Int := 252;
   END_VAR
   VAR_TEMP   // added for the SCL form of the ladder/FBD networks
      _w1 : Bool;
      _w2 : Bool;
      _w3 : Bool;
      _w4 : Bool;
      _w5 : Bool;
      _w6 : Bool;
      _w7 : Bool;
      _w8 : Bool;
      _w9 : Bool;
      _w10 : Bool;
   END_VAR
BEGIN

REGION Network 1: Reset Output Variables.
   // Variables set to zero, will be set based on current control state
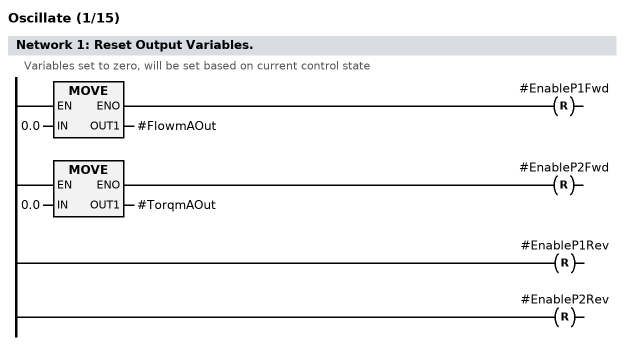
   RUNG wire#powerrail
      Move(in := 0.0, out1 => #FlowmAOut)
      R_Coil( #EnableP1Fwd )
   END_RUNG
   RUNG wire#powerrail
      Move(in := 0.0, out1 => #TorqmAOut)
      R_Coil( #EnableP2Fwd )
   END_RUNG
   RUNG wire#powerrail
      R_Coil( #EnableP1Rev )
   END_RUNG
   RUNG wire#powerrail
      R_Coil( #EnableP2Rev )
   END_RUNG
   // the same network as SCL:
   #FlowmAOut := 0.0;
   #EnableP1Fwd := FALSE;
   #TorqmAOut := 0.0;
   #EnableP2Fwd := FALSE;
   #EnableP1Rev := FALSE;
   #EnableP2Rev := FALSE;
END_REGION

REGION Network 2: Home Position and Osc Endpoints
   // On startup set current position as Zero. 
   // Adjust Home position by Bump value
   // Calculate new endpoints for oscillator. 
   // Osc Home High and Low are used for warnings while Holding positiong. Note High position is 2x Rotational Deg per count above home while low is just 1 deg per count below home
   // Note: Bump Inputs are set on HMI . If holding they will be reset when bump finished moving, if not holding reset the bits.
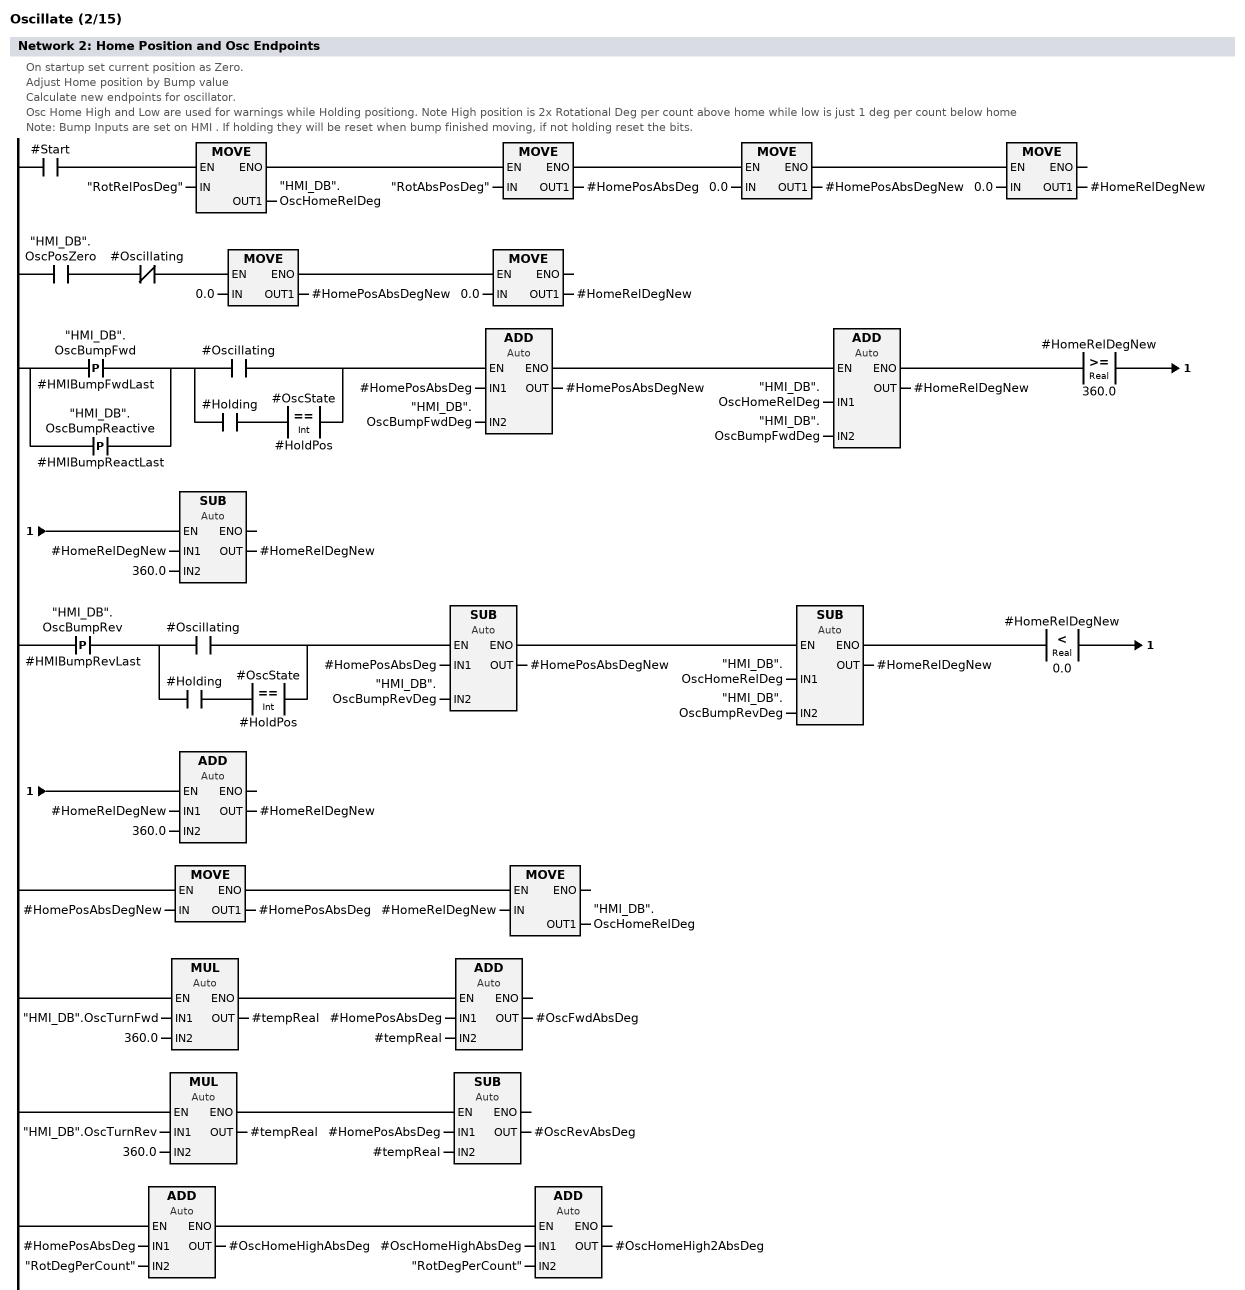
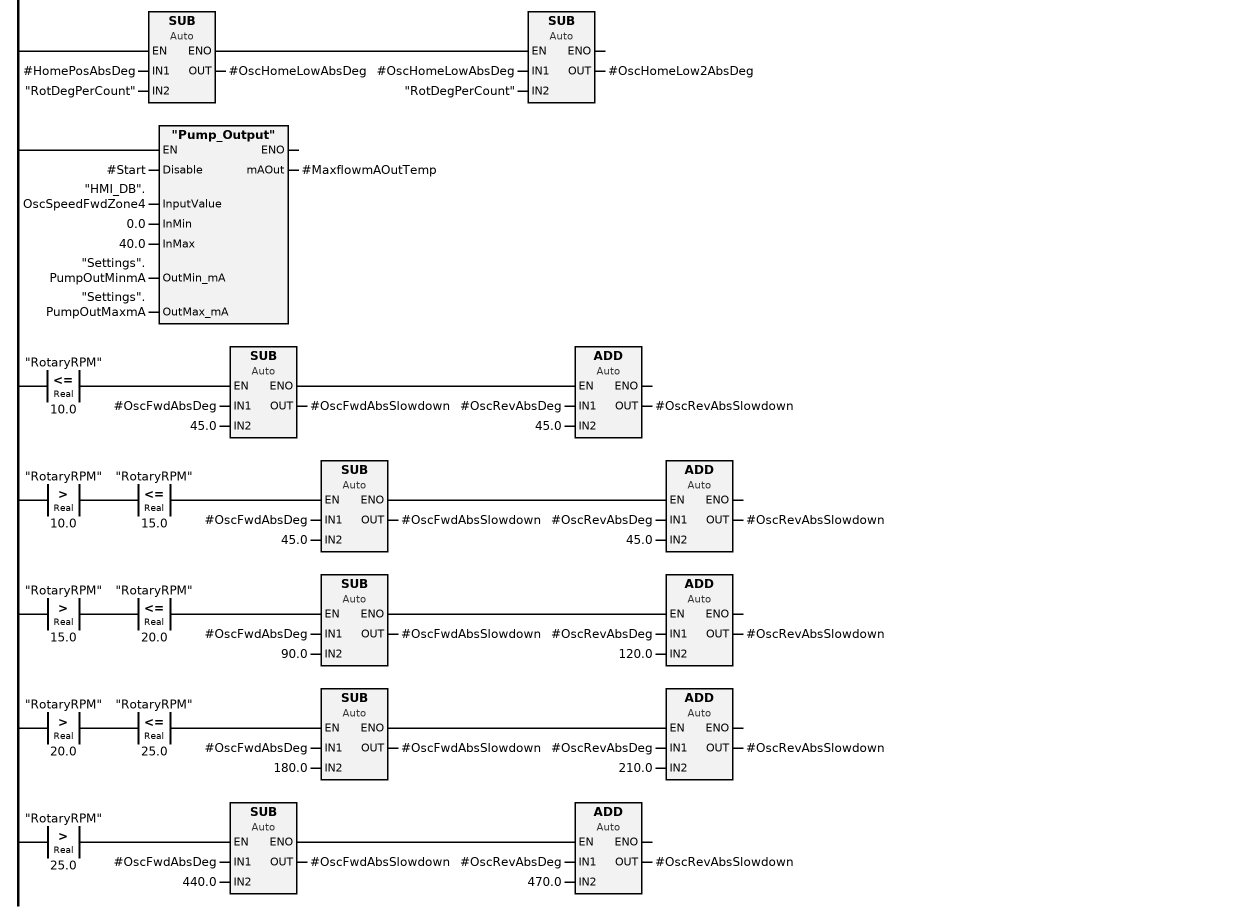
   RUNG wire#powerrail
      Contact( #Start )
      Move(in := "RotRelPosDeg", out1 => "HMI_DB".OscHomeRelDeg)
      Move(in := "RotAbsPosDeg", out1 => #HomePosAbsDeg)
      Move(in := 0.0, out1 => #HomePosAbsDegNew)
      Move(in := 0.0, out1 => #HomeRelDegNew)
   END_RUNG
   RUNG wire#powerrail
      Contact( "HMI_DB".OscPosZero )
      I_Contact( #Oscillating )
      Move(in := 0.0, out1 => #HomePosAbsDegNew)
      Move(in := 0.0, out1 => #HomeRelDegNew)
   END_RUNG
   RUNG wire#powerrail
      P_Contact(operand := "HMI_DB".OscBumpFwd, bit := #HMIBumpFwdLast)
      wire#w1
      Contact( #Oscillating )
      wire#w2
      Add(in1 := #HomePosAbsDeg, in2 := "HMI_DB".OscBumpFwdDeg, out => #HomePosAbsDegNew)
      Add(in1 := "HMI_DB".OscHomeRelDeg, in2 := "HMI_DB".OscBumpFwdDeg, out => #HomeRelDegNew)
      { S7_Templates := "SrcType := Real" } GE_Contact(in1 := #HomeRelDegNew, in2 := 360.0)
      Sub(in1 := #HomeRelDegNew, in2 := 360.0, out => #HomeRelDegNew)
   END_RUNG
   RUNG wire#powerrail
      P_Contact(operand := "HMI_DB".OscBumpReactive, bit := #HMIBumpReactLast)
   END_RUNG wire#w1
   RUNG wire#w1
      Contact( #Holding )
      { S7_Templates := "SrcType := Int" } EQ_Contact(in1 := #OscState, in2 := #HoldPos)
   END_RUNG wire#w2
   RUNG wire#powerrail
      P_Contact(operand := "HMI_DB".OscBumpRev, bit := #HMIBumpRevLast)
      wire#w3
      Contact( #Oscillating )
      wire#w4
      Sub(in1 := #HomePosAbsDeg, in2 := "HMI_DB".OscBumpRevDeg, out => #HomePosAbsDegNew)
      Sub(in1 := "HMI_DB".OscHomeRelDeg, in2 := "HMI_DB".OscBumpRevDeg, out => #HomeRelDegNew)
      { S7_Templates := "SrcType := Real" } LT_Contact(in1 := #HomeRelDegNew, in2 := 0.0)
      Add(in1 := #HomeRelDegNew, in2 := 360.0, out => #HomeRelDegNew)
   END_RUNG
   RUNG wire#w3
      Contact( #Holding )
      { S7_Templates := "SrcType := Int" } EQ_Contact(in1 := #OscState, in2 := #HoldPos)
   END_RUNG wire#w4
   RUNG wire#powerrail
      Move(in := #HomePosAbsDegNew, out1 => #HomePosAbsDeg)
      Move(in := #HomeRelDegNew, out1 => "HMI_DB".OscHomeRelDeg)
   END_RUNG
   RUNG wire#powerrail
      Mul(in1 := "HMI_DB".OscTurnFwd, in2 := 360.0, out => #tempReal)
      Add(in1 := #HomePosAbsDeg, in2 := #tempReal, out => #OscFwdAbsDeg)
   END_RUNG
   RUNG wire#powerrail
      Mul(in1 := "HMI_DB".OscTurnRev, in2 := 360.0, out => #tempReal)
      Sub(in1 := #HomePosAbsDeg, in2 := #tempReal, out => #OscRevAbsDeg)
   END_RUNG
   RUNG wire#powerrail
      Add(in1 := #HomePosAbsDeg, in2 := "RotDegPerCount", out => #OscHomeHighAbsDeg)
      Add(in1 := #OscHomeHighAbsDeg, in2 := "RotDegPerCount", out => #OscHomeHigh2AbsDeg)
   END_RUNG
   RUNG wire#powerrail
      Sub(in1 := #HomePosAbsDeg, in2 := "RotDegPerCount", out => #OscHomeLowAbsDeg)
      Sub(in1 := #OscHomeLowAbsDeg, in2 := "RotDegPerCount", out => #OscHomeLow2AbsDeg)
   END_RUNG
   RUNG wire#powerrail
      "Pump_Output"(Disable := #Start, InputValue := "HMI_DB".OscSpeedFwdZone4, InMin := 0.0, InMax := 40.0, OutMin_mA := "Settings".PumpOutMinmA, OutMax_mA := "Settings".PumpOutMaxmA, mAOut => #MaxflowmAOutTemp)
   END_RUNG
   RUNG wire#powerrail
      { S7_Templates := "SrcType := Real" } LE_Contact(in1 := "RotaryRPM", in2 := 10.0)
      Sub(in1 := #OscFwdAbsDeg, in2 := 45.0, out => #OscFwdAbsSlowdown)
      Add(in1 := #OscRevAbsDeg, in2 := 45.0, out => #OscRevAbsSlowdown)
   END_RUNG
   RUNG wire#powerrail
      { S7_Templates := "SrcType := Real" } GT_Contact(in1 := "RotaryRPM", in2 := 10.0)
      { S7_Templates := "SrcType := Real" } LE_Contact(in1 := "RotaryRPM", in2 := 15.0)
      Sub(in1 := #OscFwdAbsDeg, in2 := 45.0, out => #OscFwdAbsSlowdown)
      Add(in1 := #OscRevAbsDeg, in2 := 45.0, out => #OscRevAbsSlowdown)
   END_RUNG
   RUNG wire#powerrail
      { S7_Templates := "SrcType := Real" } GT_Contact(in1 := "RotaryRPM", in2 := 15.0)
      { S7_Templates := "SrcType := Real" } LE_Contact(in1 := "RotaryRPM", in2 := 20.0)
      Sub(in1 := #OscFwdAbsDeg, in2 := 90.0, out => #OscFwdAbsSlowdown)
      Add(in1 := #OscRevAbsDeg, in2 := 120.0, out => #OscRevAbsSlowdown)
   END_RUNG
   RUNG wire#powerrail
      { S7_Templates := "SrcType := Real" } GT_Contact(in1 := "RotaryRPM", in2 := 20.0)
      { S7_Templates := "SrcType := Real" } LE_Contact(in1 := "RotaryRPM", in2 := 25.0)
      Sub(in1 := #OscFwdAbsDeg, in2 := 180.0, out => #OscFwdAbsSlowdown)
      Add(in1 := #OscRevAbsDeg, in2 := 210.0, out => #OscRevAbsSlowdown)
   END_RUNG
   RUNG wire#powerrail
      { S7_Templates := "SrcType := Real" } GT_Contact(in1 := "RotaryRPM", in2 := 25.0)
      Sub(in1 := #OscFwdAbsDeg, in2 := 440.0, out => #OscFwdAbsSlowdown)
      Add(in1 := #OscRevAbsDeg, in2 := 470.0, out => #OscRevAbsSlowdown)
   END_RUNG
   // the same network as SCL:
   IF #Start THEN
       "HMI_DB".OscHomeRelDeg := "RotRelPosDeg";
       #HomePosAbsDeg := "RotAbsPosDeg";
       #HomePosAbsDegNew := 0.0;
       #HomeRelDegNew := 0.0;
   END_IF;
   IF "HMI_DB".OscPosZero AND NOT #Oscillating THEN
       #HomePosAbsDegNew := 0.0;
       #HomeRelDegNew := 0.0;
   END_IF;
   #_w1 := "HMI_DB".OscBumpFwd AND NOT #HMIBumpFwdLast;   // rising edge of "HMI_DB".OscBumpFwd
   #HMIBumpFwdLast := "HMI_DB".OscBumpFwd;
   #_w2 := "HMI_DB".OscBumpReactive AND NOT #HMIBumpReactLast;   // rising edge of "HMI_DB".OscBumpReactive
   #HMIBumpReactLast := "HMI_DB".OscBumpReactive;
   #_w3 := (#_w1 OR #_w2) AND (#Oscillating OR (#Holding AND (#OscState = #HoldPos)));
   IF #_w3 THEN
       #HomePosAbsDegNew := #HomePosAbsDeg + "HMI_DB".OscBumpFwdDeg;
       #HomeRelDegNew := "HMI_DB".OscHomeRelDeg + "HMI_DB".OscBumpFwdDeg;
   END_IF;
   IF #_w3 AND (#HomeRelDegNew >= 360.0) THEN #HomeRelDegNew := #HomeRelDegNew - 360.0; END_IF;
   #_w4 := "HMI_DB".OscBumpRev AND NOT #HMIBumpRevLast;   // rising edge of "HMI_DB".OscBumpRev
   #HMIBumpRevLast := "HMI_DB".OscBumpRev;
   #_w5 := #_w4 AND (#Oscillating OR (#Holding AND (#OscState = #HoldPos)));
   IF #_w5 THEN
       #HomePosAbsDegNew := #HomePosAbsDeg - "HMI_DB".OscBumpRevDeg;
       #HomeRelDegNew := "HMI_DB".OscHomeRelDeg - "HMI_DB".OscBumpRevDeg;
   END_IF;
   IF #_w5 AND (#HomeRelDegNew < 0.0) THEN #HomeRelDegNew := #HomeRelDegNew + 360.0; END_IF;
   #HomePosAbsDeg := #HomePosAbsDegNew;
   "HMI_DB".OscHomeRelDeg := #HomeRelDegNew;
   #tempReal := "HMI_DB".OscTurnFwd * 360.0;
   #OscFwdAbsDeg := #HomePosAbsDeg + #tempReal;
   #tempReal := "HMI_DB".OscTurnRev * 360.0;
   #OscRevAbsDeg := #HomePosAbsDeg - #tempReal;
   #OscHomeHighAbsDeg := #HomePosAbsDeg + "RotDegPerCount";
   #OscHomeHigh2AbsDeg := #OscHomeHighAbsDeg + "RotDegPerCount";
   #OscHomeLowAbsDeg := #HomePosAbsDeg - "RotDegPerCount";
   #OscHomeLow2AbsDeg := #OscHomeLowAbsDeg - "RotDegPerCount";
   "Pump_Output"(Disable := #Start,
                 InputValue := "HMI_DB".OscSpeedFwdZone4,
                 InMin := 0.0,
                 InMax := 40.0,
                 OutMin_mA := "Settings".PumpOutMinmA,
                 OutMax_mA := "Settings".PumpOutMaxmA,
                 mAOut => #MaxflowmAOutTemp);
   IF "RotaryRPM" <= 10.0 THEN
       #OscFwdAbsSlowdown := #OscFwdAbsDeg - 45.0;
       #OscRevAbsSlowdown := #OscRevAbsDeg + 45.0;
   END_IF;
   IF ("RotaryRPM" > 10.0) AND ("RotaryRPM" <= 15.0) THEN
       #OscFwdAbsSlowdown := #OscFwdAbsDeg - 45.0;
       #OscRevAbsSlowdown := #OscRevAbsDeg + 45.0;
   END_IF;
   IF ("RotaryRPM" > 15.0) AND ("RotaryRPM" <= 20.0) THEN
       #OscFwdAbsSlowdown := #OscFwdAbsDeg - 90.0;
       #OscRevAbsSlowdown := #OscRevAbsDeg + 120.0;
   END_IF;
   IF ("RotaryRPM" > 20.0) AND ("RotaryRPM" <= 25.0) THEN
       #OscFwdAbsSlowdown := #OscFwdAbsDeg - 180.0;
       #OscRevAbsSlowdown := #OscRevAbsDeg + 210.0;
   END_IF;
   IF "RotaryRPM" > 25.0 THEN
       #OscFwdAbsSlowdown := #OscFwdAbsDeg - 440.0;
       #OscRevAbsSlowdown := #OscRevAbsDeg + 470.0;
   END_IF;
END_REGION

REGION Network 3: Startup - State 0
   // Set State to zero if first block call
   // State Zero - Startup and set to  reset bits and go to  Waiting Cmd
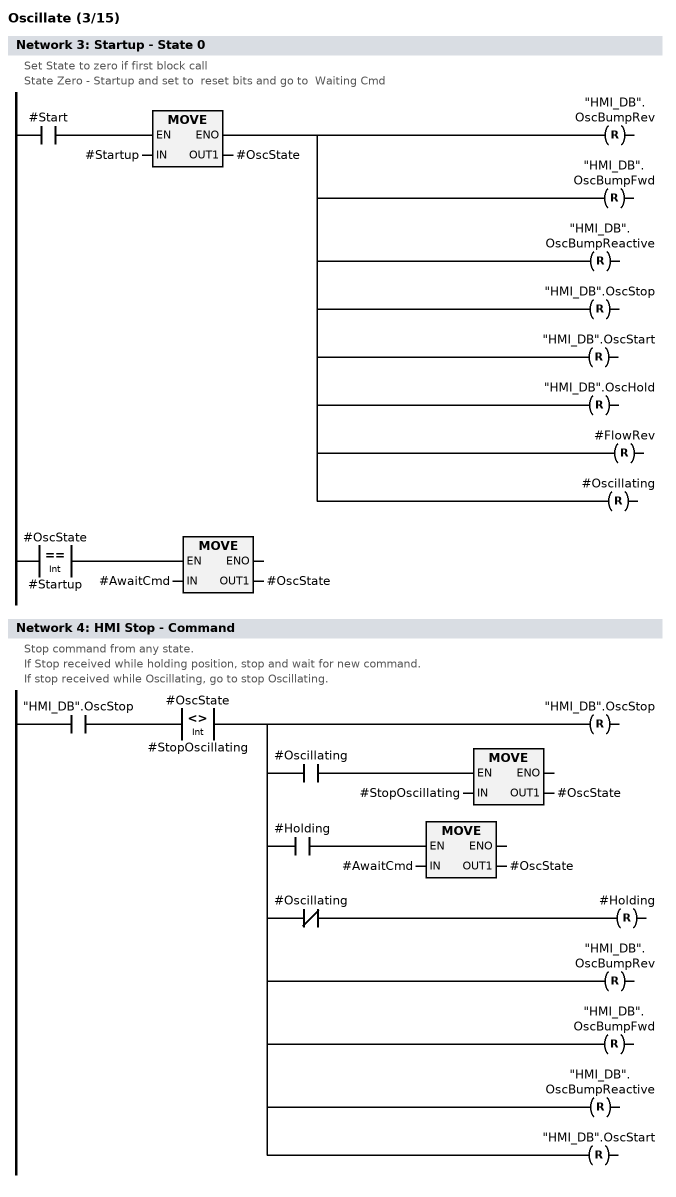
   RUNG wire#powerrail
      Contact( #Start )
      Move(in := #Startup, out1 => #OscState)
      wire#w1
      R_Coil( "HMI_DB".OscBumpRev )
   END_RUNG
   RUNG wire#w1
      R_Coil( "HMI_DB".OscBumpFwd )
   END_RUNG
   RUNG wire#w1
      R_Coil( "HMI_DB".OscBumpReactive )
   END_RUNG
   RUNG wire#w1
      R_Coil( "HMI_DB".OscStop )
   END_RUNG
   RUNG wire#w1
      R_Coil( "HMI_DB".OscStart )
   END_RUNG
   RUNG wire#w1
      R_Coil( "HMI_DB".OscHold )
   END_RUNG
   RUNG wire#w1
      R_Coil( #FlowRev )
   END_RUNG
   RUNG wire#w1
      R_Coil( #Oscillating )
   END_RUNG
   RUNG wire#powerrail
      { S7_Templates := "SrcType := Int" } EQ_Contact(in1 := #OscState, in2 := #Startup)
      Move(in := #AwaitCmd, out1 => #OscState)
   END_RUNG
   // the same network as SCL:
   IF #Start THEN
       #OscState := #Startup;
       "HMI_DB".OscBumpRev := FALSE;
       "HMI_DB".OscBumpFwd := FALSE;
       "HMI_DB".OscBumpReactive := FALSE;
       "HMI_DB".OscStop := FALSE;
       "HMI_DB".OscStart := FALSE;
       "HMI_DB".OscHold := FALSE;
       #FlowRev := FALSE;
       #Oscillating := FALSE;
   END_IF;
   IF #OscState = #Startup THEN #OscState := #AwaitCmd; END_IF;
END_REGION

REGION Network 4: HMI Stop - Command
   // Stop command from any state. 
   // If Stop received while holding position, stop and wait for new command. 
   // If stop received while Oscillating, go to stop Oscillating.
   RUNG wire#powerrail
      Contact( "HMI_DB".OscStop )
      { S7_Templates := "SrcType := Int" } NE_Contact(in1 := #OscState, in2 := #StopOscillating)
      wire#w1
      R_Coil( "HMI_DB".OscStop )
   END_RUNG
   RUNG wire#w1
      Contact( #Oscillating )
      Move(in := #StopOscillating, out1 => #OscState)
   END_RUNG
   RUNG wire#w1
      Contact( #Holding )
      Move(in := #AwaitCmd, out1 => #OscState)
   END_RUNG
   RUNG wire#w1
      I_Contact( #Oscillating )
      R_Coil( #Holding )
   END_RUNG
   RUNG wire#w1
      R_Coil( "HMI_DB".OscBumpRev )
   END_RUNG
   RUNG wire#w1
      R_Coil( "HMI_DB".OscBumpFwd )
   END_RUNG
   RUNG wire#w1
      R_Coil( "HMI_DB".OscBumpReactive )
   END_RUNG
   RUNG wire#w1
      R_Coil( "HMI_DB".OscStart )
   END_RUNG
   // the same network as SCL:
   #_w1 := "HMI_DB".OscStop AND (#OscState <> #StopOscillating);
   IF #_w1 THEN "HMI_DB".OscStop := FALSE; END_IF;
   IF #_w1 AND #Oscillating THEN #OscState := #StopOscillating; END_IF;
   IF #_w1 AND #Holding THEN #OscState := #AwaitCmd; END_IF;
   IF #_w1 AND NOT #Oscillating THEN #Holding := FALSE; END_IF;
   IF #_w1 THEN
       "HMI_DB".OscBumpRev := FALSE;
       "HMI_DB".OscBumpFwd := FALSE;
       "HMI_DB".OscBumpReactive := FALSE;
       "HMI_DB".OscStart := FALSE;
   END_IF;
END_REGION

REGION Network 5: HMI Hold - Command
   // Hold command from any state.
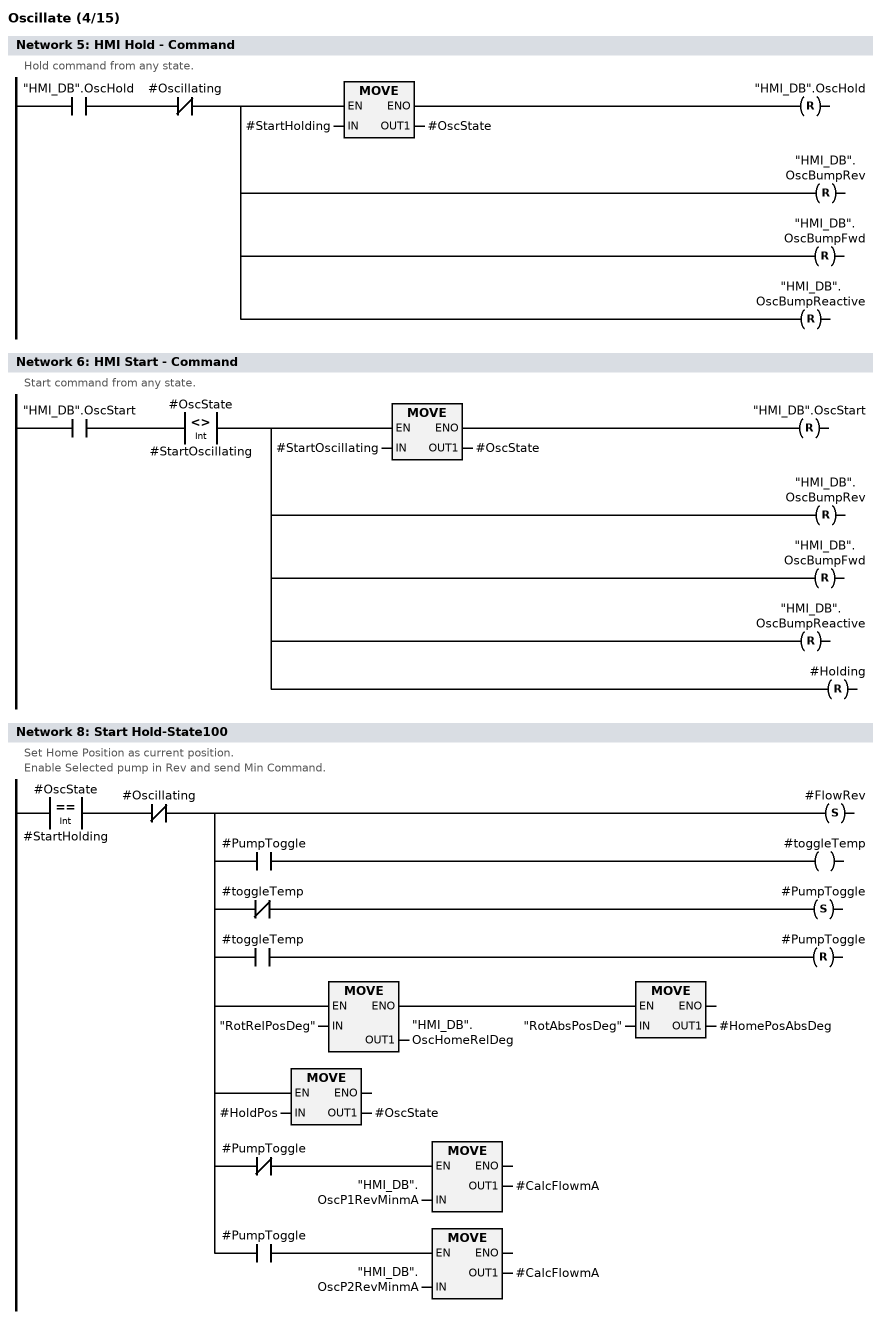
   RUNG wire#powerrail
      Contact( "HMI_DB".OscHold )
      I_Contact( #Oscillating )
      wire#w1
      Move(in := #StartHolding, out1 => #OscState)
      R_Coil( "HMI_DB".OscHold )
   END_RUNG
   RUNG wire#w1
      R_Coil( "HMI_DB".OscBumpRev )
   END_RUNG
   RUNG wire#w1
      R_Coil( "HMI_DB".OscBumpFwd )
   END_RUNG
   RUNG wire#w1
      R_Coil( "HMI_DB".OscBumpReactive )
   END_RUNG
   // the same network as SCL:
   IF "HMI_DB".OscHold AND NOT #Oscillating THEN #OscState := #StartHolding; END_IF;
   #_w1 := "HMI_DB".OscHold AND NOT #Oscillating;
   IF #_w1 THEN
       "HMI_DB".OscHold := FALSE;
       "HMI_DB".OscBumpRev := FALSE;
       "HMI_DB".OscBumpFwd := FALSE;
       "HMI_DB".OscBumpReactive := FALSE;
   END_IF;
END_REGION

REGION Network 6: HMI Start - Command
   // Start command from any state.
   RUNG wire#powerrail
      Contact( "HMI_DB".OscStart )
      { S7_Templates := "SrcType := Int" } NE_Contact(in1 := #OscState, in2 := #StartOscillating)
      wire#w1
      Move(in := #StartOscillating, out1 => #OscState)
      R_Coil( "HMI_DB".OscStart )
   END_RUNG
   RUNG wire#w1
      R_Coil( "HMI_DB".OscBumpRev )
   END_RUNG
   RUNG wire#w1
      R_Coil( "HMI_DB".OscBumpFwd )
   END_RUNG
   RUNG wire#w1
      R_Coil( "HMI_DB".OscBumpReactive )
   END_RUNG
   RUNG wire#w1
      R_Coil( #Holding )
   END_RUNG
   // the same network as SCL:
   #_w1 := "HMI_DB".OscStart AND (#OscState <> #StartOscillating);
   #_w2 := "HMI_DB".OscStart AND (#OscState <> #StartOscillating);
   IF #_w2 THEN
       #OscState := #StartOscillating;
       "HMI_DB".OscStart := FALSE;
   END_IF;
   IF #_w1 THEN
       "HMI_DB".OscBumpRev := FALSE;
       "HMI_DB".OscBumpFwd := FALSE;
       "HMI_DB".OscBumpReactive := FALSE;
       #Holding := FALSE;
   END_IF;
END_REGION

REGION Network 7: Await Cmd- State 1
   // Nothing happens in State 1 Awaiting Command- Placeholder Network if actions needed here.
END_REGION

REGION Network 8: Start Hold-State100
   // Set Home Position as current position. 
   // Enable Selected pump in Rev and send Min Command.
   RUNG wire#powerrail
      { S7_Templates := "SrcType := Int" } EQ_Contact(in1 := #OscState, in2 := #StartHolding)
      I_Contact( #Oscillating )
      wire#w1
      S_Coil( #FlowRev )
   END_RUNG
   RUNG wire#w1
      Contact( #PumpToggle )
      Coil( #toggleTemp )
   END_RUNG
   RUNG wire#w1
      I_Contact( #toggleTemp )
      S_Coil( #PumpToggle )
   END_RUNG
   RUNG wire#w1
      Contact( #toggleTemp )
      R_Coil( #PumpToggle )
   END_RUNG
   RUNG wire#w1
      Move(in := "RotRelPosDeg", out1 => "HMI_DB".OscHomeRelDeg)
      Move(in := "RotAbsPosDeg", out1 => #HomePosAbsDeg)
   END_RUNG
   RUNG wire#w1
      Move(in := #HoldPos, out1 => #OscState)
   END_RUNG
   RUNG wire#w1
      I_Contact( #PumpToggle )
      Move(in := "HMI_DB".OscP1RevMinmA, out1 => #CalcFlowmA)
   END_RUNG
   RUNG wire#w1
      Contact( #PumpToggle )
      Move(in := "HMI_DB".OscP2RevMinmA, out1 => #CalcFlowmA)
   END_RUNG
   // the same network as SCL:
   #_w1 := (#OscState = #StartHolding) AND NOT #Oscillating;
   IF #_w1 THEN #FlowRev := TRUE; END_IF;
   #toggleTemp := #_w1 AND #PumpToggle;
   IF #_w1 AND NOT #toggleTemp THEN #PumpToggle := TRUE; END_IF;
   IF #_w1 AND #toggleTemp THEN #PumpToggle := FALSE; END_IF;
   IF #_w1 THEN
       "HMI_DB".OscHomeRelDeg := "RotRelPosDeg";
       #HomePosAbsDeg := "RotAbsPosDeg";
       #OscState := #HoldPos;
   END_IF;
   IF #_w1 AND NOT #PumpToggle THEN #CalcFlowmA := "HMI_DB".OscP1RevMinmA; END_IF;
   IF #_w1 AND #PumpToggle THEN #CalcFlowmA := "HMI_DB".OscP2RevMinmA; END_IF;
END_REGION

REGION Network 9: Hold Position - State 101
   // If no Bump Received
   // - Position Held -  Maintain output
   // - Position Above home(increasing) - Stroke Hold - 
   // - Position Below Home (decreasing) - Stroke Min 
   // - Flow Rev Enabled
   // If bump received go to Bump/Reactive Bump and set new Home
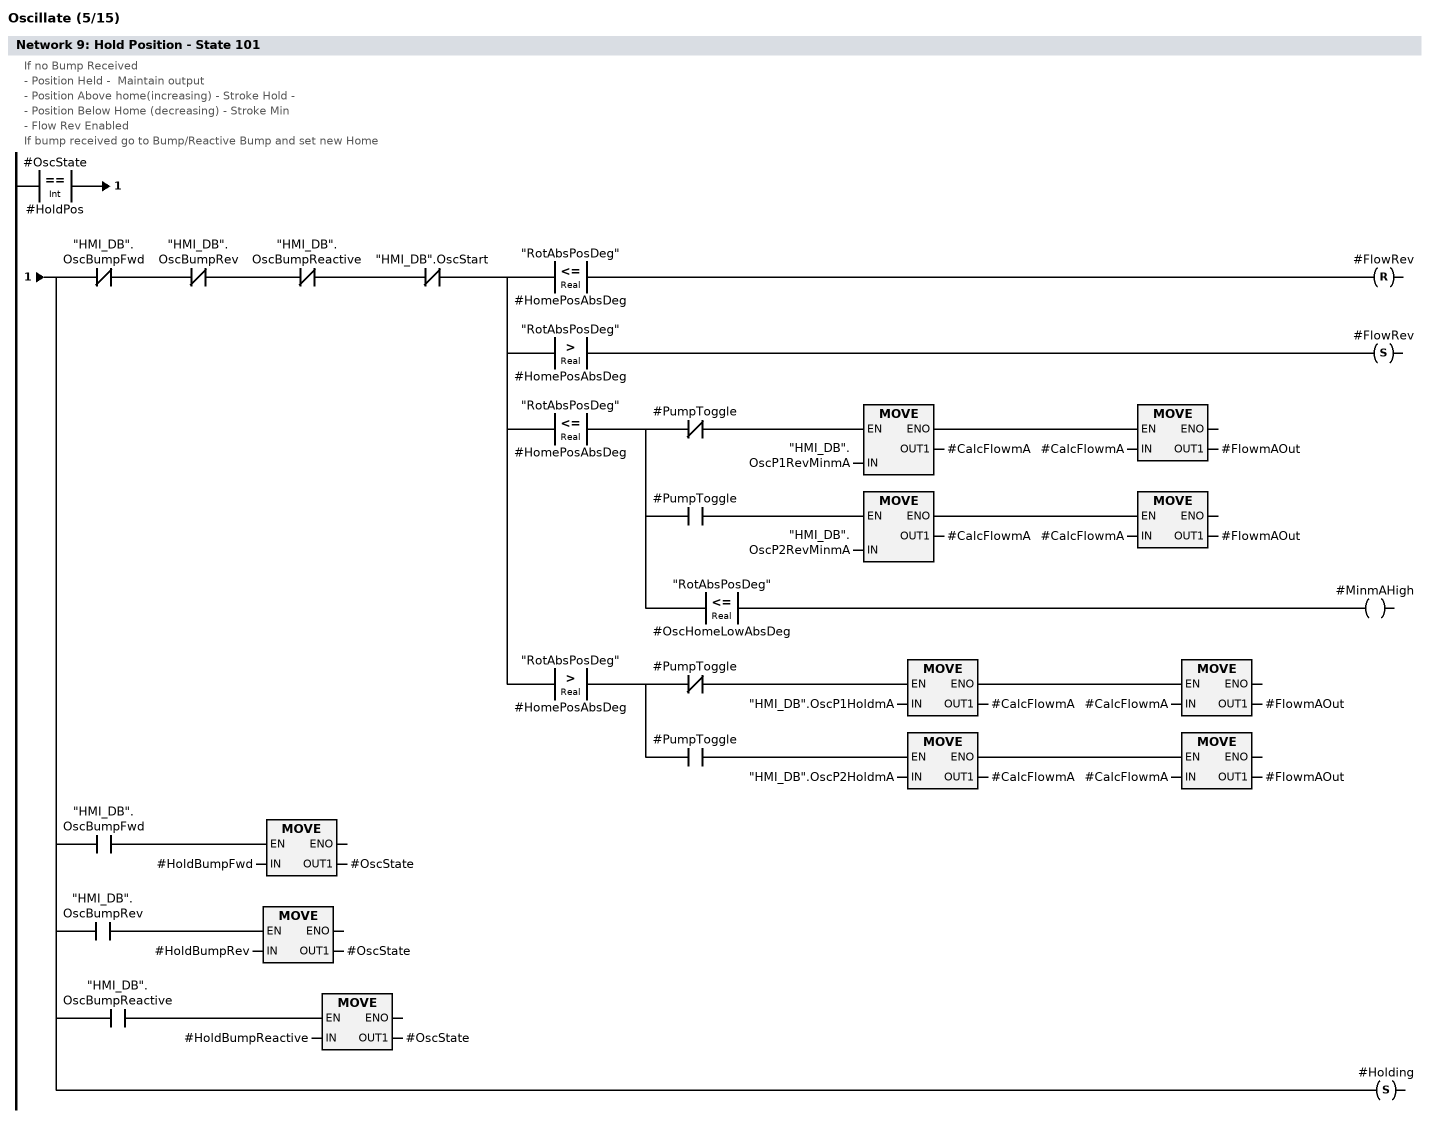
   RUNG wire#powerrail
      { S7_Templates := "SrcType := Int" } EQ_Contact(in1 := #OscState, in2 := #HoldPos)
      wire#w1
      I_Contact( "HMI_DB".OscBumpFwd )
      I_Contact( "HMI_DB".OscBumpRev )
      I_Contact( "HMI_DB".OscBumpReactive )
      I_Contact( "HMI_DB".OscStart )
      wire#w2
      { S7_Templates := "SrcType := Real" } LE_Contact(in1 := "RotAbsPosDeg", in2 := #HomePosAbsDeg)
      R_Coil( #FlowRev )
   END_RUNG
   RUNG wire#w2
      { S7_Templates := "SrcType := Real" } GT_Contact(in1 := "RotAbsPosDeg", in2 := #HomePosAbsDeg)
      S_Coil( #FlowRev )
   END_RUNG
   RUNG wire#w2
      { S7_Templates := "SrcType := Real" } LE_Contact(in1 := "RotAbsPosDeg", in2 := #HomePosAbsDeg)
      wire#w3
      I_Contact( #PumpToggle )
      Move(in := "HMI_DB".OscP1RevMinmA, out1 => #CalcFlowmA)
      Move(in := #CalcFlowmA, out1 => #FlowmAOut)
   END_RUNG
   RUNG wire#w3
      Contact( #PumpToggle )
      Move(in := "HMI_DB".OscP2RevMinmA, out1 => #CalcFlowmA)
      Move(in := #CalcFlowmA, out1 => #FlowmAOut)
   END_RUNG
   RUNG wire#w3
      { S7_Templates := "SrcType := Real" } LE_Contact(in1 := "RotAbsPosDeg", in2 := #OscHomeLowAbsDeg)
      Coil( #MinmAHigh )
   END_RUNG
   RUNG wire#w2
      { S7_Templates := "SrcType := Real" } GT_Contact(in1 := "RotAbsPosDeg", in2 := #HomePosAbsDeg)
      wire#w4
      I_Contact( #PumpToggle )
      Move(in := "HMI_DB".OscP1HoldmA, out1 => #CalcFlowmA)
      Move(in := #CalcFlowmA, out1 => #FlowmAOut)
   END_RUNG
   RUNG wire#w4
      Contact( #PumpToggle )
      Move(in := "HMI_DB".OscP2HoldmA, out1 => #CalcFlowmA)
      Move(in := #CalcFlowmA, out1 => #FlowmAOut)
   END_RUNG
   RUNG wire#w1
      Contact( "HMI_DB".OscBumpFwd )
      Move(in := #HoldBumpFwd, out1 => #OscState)
   END_RUNG
   RUNG wire#w1
      Contact( "HMI_DB".OscBumpRev )
      Move(in := #HoldBumpRev, out1 => #OscState)
   END_RUNG
   RUNG wire#w1
      Contact( "HMI_DB".OscBumpReactive )
      Move(in := #HoldBumpReactive, out1 => #OscState)
   END_RUNG
   RUNG wire#w1
      S_Coil( #Holding )
   END_RUNG
   // the same network as SCL:
   #_w1 := #OscState = #HoldPos;
   #_w2 := #_w1 AND NOT "HMI_DB".OscBumpFwd AND NOT "HMI_DB".OscBumpRev AND NOT "HMI_DB".OscBumpReactive AND NOT "HMI_DB".OscStart;
   IF #_w2 AND ("RotAbsPosDeg" <= #HomePosAbsDeg) THEN #FlowRev := FALSE; END_IF;
   IF #_w2 AND ("RotAbsPosDeg" > #HomePosAbsDeg) THEN #FlowRev := TRUE; END_IF;
   #_w3 := #_w2 AND ("RotAbsPosDeg" <= #HomePosAbsDeg);
   IF #_w3 AND NOT #PumpToggle THEN
       #CalcFlowmA := "HMI_DB".OscP1RevMinmA;
       #FlowmAOut := #CalcFlowmA;
   END_IF;
   IF #_w3 AND #PumpToggle THEN
       #CalcFlowmA := "HMI_DB".OscP2RevMinmA;
       #FlowmAOut := #CalcFlowmA;
   END_IF;
   #MinmAHigh := #_w3 AND ("RotAbsPosDeg" <= #OscHomeLowAbsDeg);
   #_w4 := #_w2 AND ("RotAbsPosDeg" > #HomePosAbsDeg);
   IF #_w4 AND NOT #PumpToggle THEN
       #CalcFlowmA := "HMI_DB".OscP1HoldmA;
       #FlowmAOut := #CalcFlowmA;
   END_IF;
   IF #_w4 AND #PumpToggle THEN
       #CalcFlowmA := "HMI_DB".OscP2HoldmA;
       #FlowmAOut := #CalcFlowmA;
   END_IF;
   IF #_w1 AND "HMI_DB".OscBumpFwd THEN #OscState := #HoldBumpFwd; END_IF;
   IF #_w1 AND "HMI_DB".OscBumpRev THEN #OscState := #HoldBumpRev; END_IF;
   IF #_w1 AND "HMI_DB".OscBumpReactive THEN #OscState := #HoldBumpReactive; END_IF;
   IF #_w1 THEN #Holding := TRUE; END_IF;
END_REGION

REGION Network 10: Hold Bump Fwd - State 102
   // Move quill to new position in the FWD direction. 
   // Start at Min and Ramp up until speed reach. 
   // If Approaching Torq Limit, limit output flow. 
   // At or above new home position, output min and hold position
   // Note: Dummy Move On Maintain speed there as visual only.
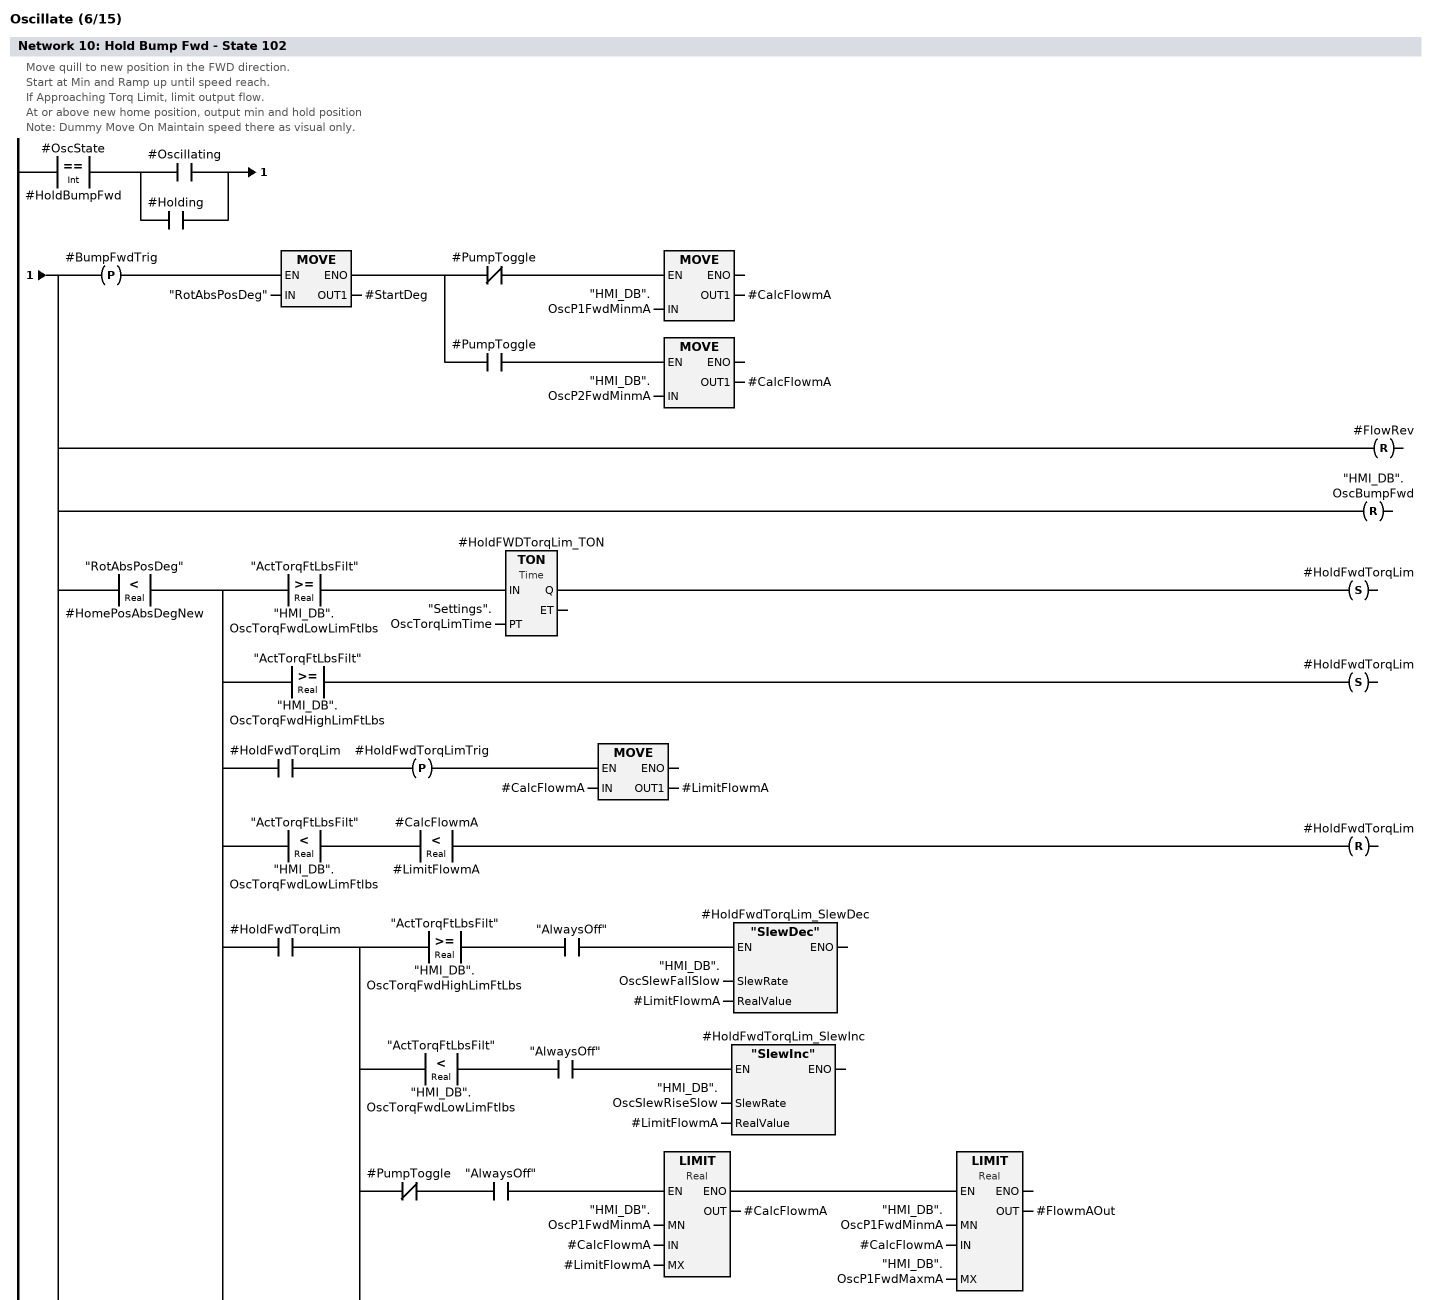
